LIN {X 0,Y 372.298,Z 1147.138,A -85,B 0,C 180,E1 19316.898,E2 19316.898} C_VEL
LIN {X 0,Y 364.057,Z 1169.224,A -85,B 0,C 180,E1 19324.16,E2 19324.16} C_VEL
LIN {X 0,Y 359.69,Z 1184.497,A -85,B 0,C 180,E1 19331.078,E2 19331.078} C_VEL
LIN {X 0,Y 357.708,Z 1194.571,A -85,B 0,C 180,E1 19337.805,E2 19337.805} C_VEL
LIN {X 0,Y 357.23,Z 1199.163,A -85,B 0,C 180,E1 19342.708,E2 19342.708} C_VEL
LIN {X 0,Y 357.403,Z 1201.877,A -85,B 0,C 180,E1 19349.999,E2 19349.999} C_VEL
LIN {X 0,Y 357.158,Z 1200.648,A -85,B 0,C 180,E1 19354.853,E2 19354.853} C_VEL
LIN {X 0,Y 357.531,Z 1196.078,A -85,B 0,C 180,E1 19360.963,E2 19360.963} C_VEL
LIN {X 0,Y 359.366,Z 1186.13,A -85,B 0,C 180,E1 19368.221,E2 19368.221} C_VEL
LIN {X 0,Y 364.091,Z 1170.43,A -85,B 0,C 180,E1 19375.834,E2 19375.834} C_VEL
LIN {X 0,Y 373.501,Z 1147.076,A -85,B 0,C 180,E1 19383.764,E2 19383.764} C_VEL
LIN {X 0,Y 386.478,Z 1119.54,A -85,B 0,C 180,E1 19390.645,E2 19390.645} C_VEL
LIN {X 0,Y 403.357,Z 1085.357,A -85,B 0,C 180,E1 19396.93,E2 19396.93} C_VEL
LIN {X 0,Y 421.007,Z 1048.766,A -85,B 0,C 180,E1 19401.873,E2 19401.873} C_VEL
LIN {X 0,Y 428.353,Z 1032.866,A -85,B 0,C 180,E1 19403.602,E2 19403.602} C_VEL
LIN {X 0,Y 431.334,Z 1020.773,A -85,B 0,C 180,E1 19405.233,E2 19405.233} C_VEL
LIN {X 0,Y 434.515,Z 1008.135,A -85,B 0,C 180,E1 19406.804,E2 19406.804} C_VEL
LIN {X 0,Y 450.973,Z 967.222,A -85,B 0,C 180,E1 19409.773,E2 19409.773} C_VEL
LIN {X 0,Y 465.114,Z 924.641,A -85,B 0,C 180,E1 19412.061,E2 19412.061} C_VEL
LIN {X 0,Y 459.039,Z 904.432,A -85,B 0,C 180,E1 19416.015,E2 19416.015} C_VEL
LIN {X 0,Y 451.558,Z 885.268,A -85,B 0,C 180,E1 19420.962,E2 19420.962} C_VEL
LIN {X 0,Y 444.782,Z 870.029,A -85,B 0,C 180,E1 19426.623,E2 19426.623} C_VEL
LIN {X 0,Y 441.283,Z 863.474,A -85,B 0,C 180,E1 19430.644,E2 19430.644} C_VEL
LIN {X 0,Y 439.558,Z 858.068,A -85,B 0,C 180,E1 19435.075,E2 19435.075} C_VEL
LIN {X 0,Y 439.377,Z 858.667,A -85,B 0,C 180,E1 19441.299,E2 19441.299} C_VEL
LIN {X 0,Y 441.594,Z 865.474,A -85,B 0,C 180,E1 19446.576,E2 19446.576} C_VEL
LIN {X 0,Y 445.757,Z 876.264,A -85,B 0,C 180,E1 19451.742,E2 19451.742} C_VEL
LIN {X 0,Y 451.62,Z 892.448,A -85,B 0,C 180,E1 19457.03,E2 19457.03} C_VEL
LIN {X 0,Y 457.495,Z 912.755,A -85,B 0,C 180,E1 19461.942,E2 19461.942} C_VEL
LIN {X 0,Y 459.188,Z 923.225,A -85,B 0,C 180,E1 19463.947,E2 19463.947} C_VEL
LIN {X 0,Y 443.527,Z 964.309,A -85,B 0,C 180,E1 19466.729,E2 19466.729} C_VEL
LIN {X 0,Y 425.31,Z 1003.875,A -85,B 0,C 180,E1 19470.42,E2 19470.42} C_VEL
LIN {X 0,Y 407.151,Z 1038.144,A -85,B 0,C 180,E1 19474.868,E2 19474.868} C_VEL
LIN {X 0,Y 390.184,Z 1067.744,A -85,B 0,C 180,E1 19480.105,E2 19480.105} C_VEL
LIN {X 0,Y 374.283,Z 1094.174,A -85,B 0,C 180,E1 19486.659,E2 19486.659} C_VEL
LIN {X 0,Y 362.655,Z 1114.122,A -85,B 0,C 180,E1 19493.626,E2 19493.626} C_VEL
LIN {X 0,Y 355.097,Z 1129.056,A -85,B 0,C 180,E1 19501.232,E2 19501.232} C_VEL
LIN {X 0,Y 351.155,Z 1138.273,A -85,B 0,C 180,E1 19508.598,E2 19508.598} C_VEL
LIN {X 0,Y 349.591,Z 1142.566,A -85,B 0,C 180,E1 19514.97,E2 19514.97} C_VEL
LIN {X 0,Y 349.351,Z 1143.375,A -85,B 0,C 180,E1 19522.545,E2 19522.545} C_VEL
LIN {X 0,Y 350.426,Z 1139.643,A -85,B 0,C 180,E1 19530.001,E2 19530.001} C_VEL
LIN {X 0,Y 352.724,Z 1131.212,A -85,B 0,C 180,E1 19537.386,E2 19537.386} C_VEL
LIN {X 0,Y 357.711,Z 1118.01,A -85,B 0,C 180,E1 19544.684,E2 19544.684} C_VEL
LIN {X 0,Y 366.523,Z 1099.034,A -85,B 0,C 180,E1 19551.782,E2 19551.782} C_VEL
LIN {X 0,Y 378.822,Z 1074.876,A -85,B 0,C 180,E1 19558.276,E2 19558.276} C_VEL
LIN {X 0,Y 394.375,Z 1044.03,A -85,B 0,C 180,E1 19564.249,E2 19564.249} C_VEL
LIN {X 0,Y 410.276,Z 1010.143,A -85,B 0,C 180,E1 19569.011,E2 19569.011} C_VEL
LIN {X 0,Y 425.898,Z 973.002,A -85,B 0,C 180,E1 19572.877,E2 19572.877} C_VEL
LIN {X 0,Y 441.528,Z 928.725,A -85,B 0,C 180,E1 19576.199,E2 19576.199} C_VEL
LIN {X 0,Y 445.75,Z 914.752,A -85,B 0,C 180,E1 19577.03,E2 19577.03} C_VEL
LIN {X 0,Y 437.347,Z 885.924,A -85,B 0,C 180,E1 19581.941,E2 19581.941} C_VEL
LIN {X 0,Y 428.04,Z 862.19,A -85,B 0,C 180,E1 19586.817,E2 19586.817} C_VEL
LIN {X 0,Y 417.98,Z 841.816,A -85,B 0,C 180,E1 19592.252,E2 19592.252} C_VEL
LIN {X 0,Y 410.472,Z 828.721,A -85,B 0,C 180,E1 19596.981,E2 19596.981} C_VEL
LIN {X 0,Y 406.667,Z 822.607,A -85,B 0,C 180,E1 19599.89,E2 19599.89} C_VEL
LIN {X 0,Y 403.865,Z 817.713,A -85,B 0,C 180,E1 19602.576,E2 19602.576} C_VEL
LIN {X 0,Y 400.692,Z 811.484,A -85,B 0,C 180,E1 19607.241,E2 19607.241} C_VEL
LIN {X 0,Y 399.55,Z 810.186,A -85,B 0,C 180,E1 19615.656,E2 19615.656} C_VEL
LIN {X 0,Y 402.264,Z 812.631,A -85,B 0,C 180,E1 19620.532,E2 19620.532} C_VEL
LIN {X 0,Y 406.945,Z 820.695,A -85,B 0,C 180,E1 19625.454,E2 19625.454} C_VEL
LIN {X 0,Y 414.067,Z 831.922,A -85,B 0,C 180,E1 19630.382,E2 19630.382} C_VEL
LIN {X 0,Y 424.174,Z 849.805,A -85,B 0,C 180,E1 19635.792,E2 19635.792} C_VEL
LIN {X 0,Y 435.914,Z 873.631,A -85,B 0,C 180,E1 19641.105,E2 19641.105} C_VEL
LIN {X 0,Y 447.798,Z 903.771,A -85,B 0,C 180,E1 19646.285,E2 19646.285} C_VEL
LIN {X 0,Y 453.221,Z 922.428,A -85,B 0,C 180,E1 19648.947,E2 19648.947} C_VEL
LIN {X 0,Y 439.542,Z 968.645,A -85,B 0,C 180,E1 19651.454,E2 19651.454} C_VEL
LIN {X 0,Y 424.425,Z 1010.952,A -85,B 0,C 180,E1 19654.623,E2 19654.623} C_VEL
LIN {X 0,Y 407,Z 1053.443,A -85,B 0,C 180,E1 19658.985,E2 19658.985} C_VEL
LIN {X 0,Y 391.108,Z 1089.121,A -85,B 0,C 180,E1 19663.978,E2 19663.978} C_VEL
LIN {X 0,Y 376.256,Z 1121.494,A -85,B 0,C 180,E1 19670.013,E2 19670.013} C_VEL
LIN {X 0,Y 364.257,Z 1148.631,A -85,B 0,C 180,E1 19676.893,E2 19676.893} C_VEL
LIN {X 0,Y 356.026,Z 1170.188,A -85,B 0,C 180,E1 19684.276,E2 19684.276} C_VEL
LIN {X 0,Y 351.536,Z 1185.408,A -85,B 0,C 180,E1 19691.659,E2 19691.659} C_VEL
LIN {X 0,Y 349.74,Z 1195.19,A -85,B 0,C 180,E1 19698.787,E2 19698.787} C_VEL
LIN {X 0,Y 349.272,Z 1199.924,A -85,B 0,C 180,E1 19705.035,E2 19705.035} C_VEL
LIN {X 0,Y 349.526,Z 1201.22,A -85,B 0,C 180,E1 19709.999,E2 19709.999} C_VEL
LIN {X 0,Y 349.229,Z 1199.679,A -85,B 0,C 180,E1 19715.66,E2 19715.66} C_VEL
LIN {X 0,Y 349.823,Z 1194.118,A -85,B 0,C 180,E1 19722.472,E2 19722.472} C_VEL
LIN {X 0,Y 352.296,Z 1183.154,A -85,B 0,C 180,E1 19730.068,E2 19730.068} C_VEL
LIN {X 0,Y 357.852,Z 1166.625,A -85,B 0,C 180,E1 19737.677,E2 19737.677} C_VEL
LIN {X 0,Y 368.006,Z 1143.362,A -85,B 0,C 180,E1 19745.45,E2 19745.45} C_VEL
LIN {X 0,Y 381.934,Z 1115.333,A -85,B 0,C 180,E1 19752.267,E2 19752.267} C_VEL
LIN {X 0,Y 399.336,Z 1081.94,A -85,B 0,C 180,E1 19758.284,E2 19758.284} C_VEL
LIN {X 0,Y 417.911,Z 1044.442,A -85,B 0,C 180,E1 19763.226,E2 19763.226} C_VEL
LIN {X 0,Y 434.515,Z 1008.135,A -85,B 0,C 180,E1 19766.804,E2 19766.804} C_VEL
LIN {X 0,Y 435.747,Z 999.983,A -85,B 0,C 180,E1 19767.933,E2 19767.933} C_VEL
LIN {X 0,Y 437.139,Z 991.635,A -85,B 0,C 180,E1 19769.014,E2 19769.014} C_VEL
LIN {X 0,Y 454.038,Z 947.387,A -85,B 0,C 180,E1 19771.825,E2 19771.825} C_VEL
LIN {X 0,Y 460.132,Z 928.064,A -85,B 0,C 180,E1 19772.848,E2 19772.848} C_VEL
LIN {X 0,Y 454.249,Z 907.989,A -85,B 0,C 180,E1 19776.996,E2 19776.996} C_VEL
LIN {X 0,Y 447.608,Z 890.491,A -85,B 0,C 180,E1 19781.808,E2 19781.808} C_VEL
LIN {X 0,Y 441.752,Z 876.873,A -85,B 0,C 180,E1 19787.158,E2 19787.158} C_VEL
LIN {X 0,Y 438.637,Z 870.605,A -85,B 0,C 180,E1 19791.212,E2 19791.212} C_VEL
LIN {X 0,Y 437.371,Z 865.682,A -85,B 0,C 180,E1 19795.05,E2 19795.05} C_VEL
LIN {X 0,Y 437.168,Z 865.729,A -85,B 0,C 180,E1 19800.872,E2 19800.872} C_VEL
LIN {X 0,Y 439.014,Z 873.18,A -85,B 0,C 180,E1 19806.615,E2 19806.615} C_VEL
LIN {X 0,Y 443.01,Z 884.158,A -85,B 0,C 180,E1 19811.816,E2 19811.816} C_VEL
LIN {X 0,Y 448.428,Z 900.54,A -85,B 0,C 180,E1 19817.155,E2 19817.155} C_VEL
LIN {X 0,Y 453.305,Z 919.811,A -85,B 0,C 180,E1 19821.836,E2 19821.836} C_VEL
LIN {X 0,Y 454.599,Z 925.88,A -85,B 0,C 180,E1 19823.12,E2 19823.12} C_VEL
LIN {X 0,Y 438.258,Z 967.608,A -85,B 0,C 180,E1 19826.048,E2 19826.048} C_VEL
LIN {X 0,Y 420.056,Z 1005.918,A -85,B 0,C 180,E1 19829.672,E2 19829.672} C_VEL
LIN {X 0,Y 400.332,Z 1041.744,A -85,B 0,C 180,E1 19834.425,E2 19834.425} C_VEL
LIN {X 0,Y 382.656,Z 1071.18,A -85,B 0,C 180,E1 19839.854,E2 19839.854} C_VEL
LIN {X 0,Y 366.795,Z 1096.673,A -85,B 0,C 180,E1 19846.409,E2 19846.409} C_VEL
LIN {X 0,Y 355.017,Z 1115.873,A -85,B 0,C 180,E1 19853.424,E2 19853.424} C_VEL
LIN {X 0,Y 347.124,Z 1130.81,A -85,B 0,C 180,E1 19861.39,E2 19861.39} C_VEL
LIN {X 0,Y 343.082,Z 1139.88,A -85,B 0,C 180,E1 19869.369,E2 19869.369} C_VEL
LIN {X 0,Y 341.489,Z 1144.054,A -85,B 0,C 180,E1 19877.218,E2 19877.218} C_VEL
LIN {X 0,Y 341.718,Z 1143.309,A -85,B 0,C 180,E1 19884.927,E2 19884.927} C_VEL
LIN {X 0,Y 342.88,Z 1139.282,A -85,B 0,C 180,E1 19891.264,E2 19891.264} C_VEL
LIN {X 0,Y 345.586,Z 1130.291,A -85,B 0,C 180,E1 19898.805,E2 19898.805} C_VEL
LIN {X 0,Y 351.36,Z 1116.165,A -85,B 0,C 180,E1 19906.235,E2 19906.235} C_VEL
LIN {X 0,Y 361.614,Z 1095.823,A -85,B 0,C 180,E1 19913.62,E2 19913.62} C_VEL
LIN {X 0,Y 376.074,Z 1068.411,A -85,B 0,C 180,E1 19920.552,E2 19920.552} C_VEL
LIN {X 0,Y 391.531,Z 1038.192,A -85,B 0,C 180,E1 19926.058,E2 19926.058} C_VEL
LIN {X 0,Y 408.575,Z 1002.491,A -85,B 0,C 180,E1 19930.799,E2 19930.799} C_VEL
LIN {X 0,Y 425.037,Z 962.822,A -85,B 0,C 180,E1 19934.608,E2 19934.608} C_VEL
LIN {X 0,Y 438.935,Z 922.777,A -85,B 0,C 180,E1 19937.426,E2 19937.426} C_VEL
LIN {X 0,Y 439.949,Z 917.005,A -85,B 0,C 180,E1 19937.907,E2 19937.907} C_VEL
LIN {X 0,Y 432.477,Z 890.045,A -85,B 0,C 180,E1 19942.663,E2 19942.663} C_VEL
LIN {X 0,Y 423.57,Z 866.773,A -85,B 0,C 180,E1 19947.639,E2 19947.639} C_VEL
LIN {X 0,Y 414.395,Z 847.583,A -85,B 0,C 180,E1 19952.992,E2 19952.992} C_VEL
LIN {X 0,Y 407.812,Z 835.438,A -85,B 0,C 180,E1 19957.505,E2 19957.505} C_VEL
LIN {X 0,Y 402.53,Z 825.678,A -85,B 0,C 180,E1 19962.396,E2 19962.396} C_VEL
LIN {X 0,Y 399.093,Z 819.165,A -85,B 0,C 180,E1 19967.418,E2 19967.418} C_VEL
LIN {X 0,Y 398.181,Z 817.941,A -85,B 0,C 180,E1 19975.641,E2 19975.641} C_VEL
LIN {X 0,Y 400.691,Z 820.234,A -85,B 0,C 180,E1 19980.332,E2 19980.332} C_VEL
LIN {X 0,Y 405.241,Z 828.467,A -85,B 0,C 180,E1 19985.343,E2 19985.343} C_VEL
LIN {X 0,Y 411.935,Z 839.468,A -85,B 0,C 180,E1 19990.163,E2 19990.163} C_VEL
LIN {X 0,Y 421.528,Z 857.101,A -85,B 0,C 180,E1 19995.546,E2 19995.546} C_VEL
LIN {X 0,Y 432.262,Z 880.049,A -85,B 0,C 180,E1 20000.724,E2 20000.724} C_VEL
LIN {X 0,Y 442.967,Z 908.697,A -85,B 0,C 180,E1 20005.777,E2 20005.777} C_VEL
LIN {X 0,Y 447.647,Z 925.803,A -85,B 0,C 180,E1 20008.28,E2 20008.28} C_VEL
LIN {X 0,Y 434.055,Z 970.322,A -85,B 0,C 180,E1 20010.742,E2 20010.742} C_VEL
LIN {X 0,Y 418.224,Z 1012.969,A -85,B 0,C 180,E1 20013.996,E2 20013.996} C_VEL
LIN {X 0,Y 400.743,Z 1054.371,A -85,B 0,C 180,E1 20018.319,E2 20018.319} C_VEL
LIN {X 0,Y 383.631,Z 1091.344,A -85,B 0,C 180,E1 20023.632,E2 20023.632} C_VEL
LIN {X 0,Y 368.518,Z 1123.103,A -85,B 0,C 180,E1 20029.77,E2 20029.77} C_VEL
LIN {X 0,Y 355.85,Z 1150.918,A -85,B 0,C 180,E1 20037.127,E2 20037.127} C_VEL
LIN {X 0,Y 347.601,Z 1171.912,A -85,B 0,C 180,E1 20044.813,E2 20044.813} C_VEL
LIN {X 0,Y 343.236,Z 1187.034,A -85,B 0,C 180,E1 20052.711,E2 20052.711} C_VEL
LIN {X 0,Y 341.724,Z 1195.789,A -85,B 0,C 180,E1 20059.81,E2 20059.81} C_VEL
LIN {X 0,Y 341.456,Z 1200.202,A -85,B 0,C 180,E1 20067.462,E2 20067.462} C_VEL
LIN {X 0,Y 341.586,Z 1200.233,A -85,B 0,C 180,E1 20072.534,E2 20072.534} C_VEL
LIN {X 0,Y 341.687,Z 1196.101,A -85,B 0,C 180,E1 20080.188,E2 20080.188} C_VEL
LIN {X 0,Y 343.45,Z 1186.747,A -85,B 0,C 180,E1 20087.937,E2 20087.937} C_VEL
LIN {X 0,Y 348.573,Z 1170.894,A -85,B 0,C 180,E1 20096.29,E2 20096.29} C_VEL
LIN {X 0,Y 358.125,Z 1149.375,A -85,B 0,C 180,E1 20104.223,E2 20104.223} C_VEL
LIN {X 0,Y 372.851,Z 1120.635,A -85,B 0,C 180,E1 20111.882,E2 20111.882} C_VEL
LIN {X 0,Y 390.029,Z 1088.483,A -85,B 0,C 180,E1 20118.07,E2 20118.07} C_VEL
LIN {X 0,Y 409.11,Z 1052.094,A -85,B 0,C 180,E1 20123.231,E2 20123.231} C_VEL
LIN {X 0,Y 429.335,Z 1009.589,A -85,B 0,C 180,E1 20127.571,E2 20127.571} C_VEL
LIN {X 0,Y 437.139,Z 991.635,A -85,B 0,C 180,E1 20129.014,E2 20129.014} C_VEL
LIN {X 0,Y 440.785,Z 978.212,A -85,B 0,C 180,E1 20130.407,E2 20130.407} C_VEL
LIN {X 0,Y 444.102,Z 964.397,A -85,B 0,C 180,E1 20131.741,E2 20131.741} C_VEL
LIN {X 0,Y 455.353,Z 932.19,A -85,B 0,C 180,E1 20133.536,E2 20133.536} C_VEL
LIN {X 0,Y 449.837,Z 912.417,A -85,B 0,C 180,E1 20137.8,E2 20137.8} C_VEL
LIN {X 0,Y 443.79,Z 895.75,A -85,B 0,C 180,E1 20142.62,E2 20142.62} C_VEL
LIN {X 0,Y 438.305,Z 882.887,A -85,B 0,C 180,E1 20148.067,E2 20148.067} C_VEL
LIN {X 0,Y 436.988,Z 879.284,A -85,B 0,C 180,E1 20150.049,E2 20150.049} C_VEL
LIN {X 0,Y 434.727,Z 873.097,A -85,B 0,C 180,E1 20156.019,E2 20156.019} C_VEL
LIN {X 0,Y 434.664,Z 873.589,A -85,B 0,C 180,E1 20161.002,E2 20161.002} C_VEL
LIN {X 0,Y 436.602,Z 881.447,A -85,B 0,C 180,E1 20166.964,E2 20166.964} C_VEL
LIN {X 0,Y 440.476,Z 893.236,A -85,B 0,C 180,E1 20172.387,E2 20172.387} C_VEL
LIN {X 0,Y 445.54,Z 910.373,A -85,B 0,C 180,E1 20177.779,E2 20177.779} C_VEL
LIN {X 0,Y 449.726,Z 929.919,A -85,B 0,C 180,E1 20182.394,E2 20182.394} C_VEL
LIN {X 0,Y 432.01,Z 973.227,A -85,B 0,C 180,E1 20185.539,E2 20185.539} C_VEL
LIN {X 0,Y 413.804,Z 1009.781,A -85,B 0,C 180,E1 20189.127,E2 20189.127} C_VEL
LIN {X 0,Y 393.687,Z 1045.079,A -85,B 0,C 180,E1 20193.925,E2 20193.925} C_VEL
LIN {X 0,Y 374.913,Z 1074.943,A -85,B 0,C 180,E1 20199.665,E2 20199.665} C_VEL
LIN {X 0,Y 359.807,Z 1098.302,A -85,B 0,C 180,E1 20205.893,E2 20205.893} C_VEL
LIN {X 0,Y 346.94,Z 1118.402,A -85,B 0,C 180,E1 20213.565,E2 20213.565} C_VEL
LIN {X 0,Y 339.767,Z 1131.284,A -85,B 0,C 180,E1 20220.712,E2 20220.712} C_VEL
LIN {X 0,Y 335.363,Z 1140.424,A -85,B 0,C 180,E1 20228.872,E2 20228.872} C_VEL
LIN {X 0,Y 333.656,Z 1144.679,A -85,B 0,C 180,E1 20236.913,E2 20236.913} C_VEL
LIN {X 0,Y 333.835,Z 1143.99,A -85,B 0,C 180,E1 20244.871,E2 20244.871} C_VEL
LIN {X 0,Y 335.028,Z 1140.06,A -85,B 0,C 180,E1 20251.294,E2 20251.294} C_VEL
LIN {X 0,Y 337.826,Z 1131.151,A -85,B 0,C 180,E1 20259.008,E2 20259.008} C_VEL
LIN {X 0,Y 343.861,Z 1117.149,A -85,B 0,C 180,E1 20266.599,E2 20266.599} C_VEL
LIN {X 0,Y 354.073,Z 1097.564,A -85,B 0,C 180,E1 20273.92,E2 20273.92} C_VEL
LIN {X 0,Y 367.729,Z 1072.531,A -85,B 0,C 180,E1 20280.532,E2 20280.532} C_VEL
LIN {X 0,Y 383.67,Z 1042.925,A -85,B 0,C 180,E1 20286.215,E2 20286.215} C_VEL
LIN {X 0,Y 401.682,Z 1006.468,A -85,B 0,C 180,E1 20291.243,E2 20291.243} C_VEL
LIN {X 0,Y 417.381,Z 970.33,A -85,B 0,C 180,E1 20294.875,E2 20294.875} C_VEL
LIN {X 0,Y 433.244,Z 927.056,A -85,B 0,C 180,E1 20298.059,E2 20298.059} C_VEL
LIN {X 0,Y 434.663,Z 921.259,A -85,B 0,C 180,E1 20298.476,E2 20298.476} C_VEL
LIN {X 0,Y 427.695,Z 894.542,A -85,B 0,C 180,E1 20303.349,E2 20303.349} C_VEL
LIN {X 0,Y 419.208,Z 871.284,A -85,B 0,C 180,E1 20308.48,E2 20308.48} C_VEL
LIN {X 0,Y 409.774,Z 850.757,A -85,B 0,C 180,E1 20314.535,E2 20314.535} C_VEL
LIN {X 0,Y 403.123,Z 838.446,A -85,B 0,C 180,E1 20319.806,E2 20319.806} C_VEL
LIN {X 0,Y 399.952,Z 832.552,A -85,B 0,C 180,E1 20323.261,E2 20323.261} C_VEL
LIN {X 0,Y 397.62,Z 826.94,A -85,B 0,C 180,E1 20327.371,E2 20327.371} C_VEL
LIN {X 0,Y 396.681,Z 825.691,A -85,B 0,C 180,E1 20335.624,E2 20335.624} C_VEL
LIN {X 0,Y 399.061,Z 828.056,A -85,B 0,C 180,E1 20340.208,E2 20340.208} C_VEL
LIN {X 0,Y 403.293,Z 835.821,A -85,B 0,C 180,E1 20345.032,E2 20345.032} C_VEL
LIN {X 0,Y 409.418,Z 846.53,A -85,B 0,C 180,E1 20349.823,E2 20349.823} C_VEL
LIN {X 0,Y 418.491,Z 864.046,A -85,B 0,C 180,E1 20355.238,E2 20355.238} C_VEL
LIN {X 0,Y 428.465,Z 886.467,A -85,B 0,C 180,E1 20360.376,E2 20360.376} C_VEL
LIN {X 0,Y 438.653,Z 915.128,A -85,B 0,C 180,E1 20365.501,E2 20365.501} C_VEL
LIN {X 0,Y 442.302,Z 928.026,A -85,B 0,C 180,E1 20367.514,E2 20367.514} C_VEL
LIN {X 0,Y 428.363,Z 972.775,A -85,B 0,C 180,E1 20370.058,E2 20370.058} C_VEL
LIN {X 0,Y 411.337,Z 1016.852,A -85,B 0,C 180,E1 20373.528,E2 20373.528} C_VEL
LIN {X 0,Y 393.953,Z 1056.364,A -85,B 0,C 180,E1 20377.775,E2 20377.775} C_VEL
LIN {X 0,Y 376.276,Z 1093.339,A -85,B 0,C 180,E1 20383.232,E2 20383.232} C_VEL
LIN {X 0,Y 361.11,Z 1124.016,A -85,B 0,C 180,E1 20389.366,E2 20389.366} C_VEL
LIN {X 0,Y 348.271,Z 1151.29,A -85,B 0,C 180,E1 20396.783,E2 20396.783} C_VEL
LIN {X 0,Y 340.042,Z 1171.302,A -85,B 0,C 180,E1 20404.322,E2 20404.322} C_VEL
LIN {X 0,Y 335.469,Z 1186.262,A -85,B 0,C 180,E1 20412.297,E2 20412.297} C_VEL
LIN {X 0,Y 333.852,Z 1195.074,A -85,B 0,C 180,E1 20419.568,E2 20419.568} C_VEL
LIN {X 0,Y 333.57,Z 1199.545,A -85,B 0,C 180,E1 20427.402,E2 20427.402} C_VEL
LIN {X 0,Y 333.694,Z 1199.587,A -85,B 0,C 180,E1 20432.594,E2 20432.594} C_VEL
LIN {X 0,Y 333.803,Z 1195.472,A -85,B 0,C 180,E1 20440.431,E2 20440.431} C_VEL
LIN {X 0,Y 335.706,Z 1186.151,A -85,B 0,C 180,E1 20448.365,E2 20448.365} C_VEL
LIN {X 0,Y 340.633,Z 1171.567,A -85,B 0,C 180,E1 20456.334,E2 20456.334} C_VEL
LIN {X 0,Y 349.937,Z 1151.511,A -85,B 0,C 180,E1 20464.15,E2 20464.15} C_VEL
LIN {X 0,Y 364.606,Z 1123.772,A -85,B 0,C 180,E1 20471.894,E2 20471.894} C_VEL
LIN {X 0,Y 382.005,Z 1092.753,A -85,B 0,C 180,E1 20478.209,E2 20478.209} C_VEL
LIN {X 0,Y 402.627,Z 1054.801,A -85,B 0,C 180,E1 20483.795,E2 20483.795} C_VEL
LIN {X 0,Y 422.262,Z 1015.331,A -85,B 0,C 180,E1 20487.97,E2 20487.97} C_VEL
LIN {X 0,Y 440.817,Z 972.947,A -85,B 0,C 180,E1 20491.21,E2 20491.21} C_VEL
LIN {X 0,Y 444.102,Z 964.397,A -85,B 0,C 180,E1 20491.741,E2 20491.741} C_VEL
LIN {X 0,Y 448.813,Z 949.442,A -85,B 0,C 180,E1 20492.813,E2 20492.813} C_VEL
LIN {X 0,Y 450.391,Z 936.31,A -85,B 0,C 180,E1 20494.285,E2 20494.285} C_VEL
LIN {X 0,Y 445.385,Z 916.928,A -85,B 0,C 180,E1 20498.614,E2 20498.614} C_VEL
LIN {X 0,Y 439.799,Z 900.879,A -85,B 0,C 180,E1 20503.487,E2 20503.487} C_VEL
LIN {X 0,Y 435.77,Z 890.558,A -85,B 0,C 180,E1 20507.996,E2 20507.996} C_VEL
LIN {X 0,Y 433.138,Z 884.863,A -85,B 0,C 180,E1 20511.983,E2 20511.983} C_VEL
LIN {X 0,Y 432.186,Z 880.636,A -85,B 0,C 180,E1 20515.996,E2 20515.996} C_VEL
LIN {X 0,Y 432.089,Z 881.213,A -85,B 0,C 180,E1 20521.008,E2 20521.008} C_VEL
LIN {X 0,Y 433.788,Z 889.019,A -85,B 0,C 180,E1 20527.009,E2 20527.009} C_VEL
LIN {X 0,Y 437.424,Z 901.023,A -85,B 0,C 180,E1 20532.475,E2 20532.475} C_VEL
LIN {X 0,Y 441.708,Z 917.444,A -85,B 0,C 180,E1 20537.656,E2 20537.656} C_VEL
LIN {X 0,Y 444.85,Z 934.711,A -85,B 0,C 180,E1 20541.817,E2 20541.817} C_VEL
LIN {X 0,Y 426.821,Z 976.648,A -85,B 0,C 180,E1 20544.839,E2 20544.839} C_VEL
LIN {X 0,Y 407.57,Z 1013.666,A -85,B 0,C 180,E1 20548.568,E2 20548.568} C_VEL
LIN {X 0,Y 387.932,Z 1046.943,A -85,B 0,C 180,E1 20553.185,E2 20553.185} C_VEL
LIN {X 0,Y 368.056,Z 1077.361,A -85,B 0,C 180,E1 20559.16,E2 20559.16} C_VEL
LIN {X 0,Y 352.488,Z 1100.34,A -85,B 0,C 180,E1 20565.517,E2 20565.517} C_VEL
LIN {X 0,Y 339.415,Z 1119.989,A -85,B 0,C 180,E1 20573.276,E2 20573.276} C_VEL
LIN {X 0,Y 331.338,Z 1133.583,A -85,B 0,C 180,E1 20581.39,E2 20581.39} C_VEL
LIN {X 0,Y 327.695,Z 1140.968,A -85,B 0,C 180,E1 20588.353,E2 20588.353} C_VEL
LIN {X 0,Y 325.795,Z 1145.367,A -85,B 0,C 180,E1 20596.955,E2 20596.955} C_VEL
LIN {X 0,Y 325.92,Z 1144.724,A -85,B 0,C 180,E1 20604.681,E2 20604.681} C_VEL
LIN {X 0,Y 327.188,Z 1140.837,A -85,B 0,C 180,E1 20611.325,E2 20611.325} C_VEL
LIN {X 0,Y 330.096,Z 1132.003,A -85,B 0,C 180,E1 20619.221,E2 20619.221} C_VEL
LIN {X 0,Y 336.348,Z 1118.138,A -85,B 0,C 180,E1 20626.981,E2 20626.981} C_VEL
LIN {X 0,Y 346.944,Z 1098.638,A -85,B 0,C 180,E1 20634.444,E2 20634.444} C_VEL
LIN {X 0,Y 361.125,Z 1073.642,A -85,B 0,C 180,E1 20641.188,E2 20641.188} C_VEL
LIN {X 0,Y 377.447,Z 1044.355,A -85,B 0,C 180,E1 20646.909,E2 20646.909} C_VEL
LIN {X 0,Y 395.856,Z 1008.158,A -85,B 0,C 180,E1 20651.97,E2 20651.97} C_VEL
LIN {X 0,Y 412.103,Z 971.95,A -85,B 0,C 180,E1 20655.655,E2 20655.655} C_VEL
LIN {X 0,Y 428.557,Z 928.256,A -85,B 0,C 180,E1 20658.884,E2 20658.884} C_VEL
LIN {X 0,Y 429.331,Z 925.06,A -85,B 0,C 180,E1 20659.134,E2 20659.134} C_VEL
LIN {X 0,Y 423.055,Z 899.725,A -85,B 0,C 180,E1 20663.88,E2 20663.88} C_VEL
LIN {X 0,Y 415.512,Z 877.431,A -85,B 0,C 180,E1 20668.946,E2 20668.946} C_VEL
LIN {X 0,Y 406.688,Z 857.32,A -85,B 0,C 180,E1 20675.037,E2 20675.037} C_VEL
LIN {X 0,Y 400.812,Z 845.659,A -85,B 0,C 180,E1 20680.158,E2 20680.158} C_VEL
LIN {X 0,Y 397.955,Z 840.105,A -85,B 0,C 180,E1 20683.411,E2 20683.411} C_VEL
LIN {X 0,Y 395.639,Z 834.469,A -85,B 0,C 180,E1 20687.867,E2 20687.867} C_VEL
LIN {X 0,Y 395.316,Z 833.614,A -85,B 0,C 180,E1 20696.207,E2 20696.207} C_VEL
LIN {X 0,Y 397.334,Z 835.775,A -85,B 0,C 180,E1 20700.066,E2 20700.066} C_VEL
LIN {X 0,Y 401.176,Z 843.382,A -85,B 0,C 180,E1 20704.856,E2 20704.856} C_VEL
LIN {X 0,Y 407.172,Z 854.232,A -85,B 0,C 180,E1 20709.676,E2 20709.676} C_VEL
LIN {X 0,Y 415.57,Z 871.287,A -85,B 0,C 180,E1 20715.01,E2 20715.01} C_VEL
LIN {X 0,Y 425.149,Z 894.141,A -85,B 0,C 180,E1 20720.271,E2 20720.271} C_VEL
LIN {X 0,Y 434.473,Z 922.544,A -85,B 0,C 180,E1 20725.398,E2 20725.398} C_VEL
LIN {X 0,Y 436.687,Z 932.573,A -85,B 0,C 180,E1 20726.903,E2 20726.903} C_VEL
LIN {X 0,Y 422.714,Z 975.019,A -85,B 0,C 180,E1 20729.359,E2 20729.359} C_VEL
LIN {X 0,Y 405.188,Z 1018.977,A -85,B 0,C 180,E1 20732.878,E2 20732.878} C_VEL
LIN {X 0,Y 387.772,Z 1057.184,A -85,B 0,C 180,E1 20737.069,E2 20737.069} C_VEL
LIN {X 0,Y 369.562,Z 1094.076,A -85,B 0,C 180,E1 20742.605,E2 20742.605} C_VEL
LIN {X 0,Y 353.972,Z 1124.429,A -85,B 0,C 180,E1 20748.827,E2 20748.827} C_VEL
LIN {X 0,Y 340.81,Z 1151.385,A -85,B 0,C 180,E1 20756.34,E2 20756.34} C_VEL
LIN {X 0,Y 332.033,Z 1171.915,A -85,B 0,C 180,E1 20764.381,E2 20764.381} C_VEL
LIN {X 0,Y 327.492,Z 1186.538,A -85,B 0,C 180,E1 20772.545,E2 20772.545} C_VEL
LIN {X 0,Y 325.982,Z 1194.353,A -85,B 0,C 180,E1 20779.313,E2 20779.313} C_VEL
LIN {X 0,Y 325.707,Z 1198.888,A -85,B 0,C 180,E1 20787.339,E2 20787.339} C_VEL
LIN {X 0,Y 325.822,Z 1198.943,A -85,B 0,C 180,E1 20792.657,E2 20792.657} C_VEL
LIN {X 0,Y 325.924,Z 1194.845,A -85,B 0,C 180,E1 20800.686,E2 20800.686} C_VEL
LIN {X 0,Y 327.455,Z 1187.456,A -85,B 0,C 180,E1 20807.454,E2 20807.454} C_VEL
LIN {X 0,Y 332.047,Z 1173.866,A -85,B 0,C 180,E1 20815.615,E2 20815.615} C_VEL
LIN {X 0,Y 342.046,Z 1152.823,A -85,B 0,C 180,E1 20824.282,E2 20824.282} C_VEL
LIN {X 0,Y 356.258,Z 1127.047,A -85,B 0,C 180,E1 20831.881,E2 20831.881} C_VEL
LIN {X 0,Y 374.695,Z 1095.485,A -85,B 0,C 180,E1 20838.607,E2 20838.607} C_VEL
LIN {X 0,Y 394.502,Z 1060.417,A -85,B 0,C 180,E1 20844.001,E2 20844.001} C_VEL
LIN {X 0,Y 414.889,Z 1021.729,A -85,B 0,C 180,E1 20848.315,E2 20848.315} C_VEL
LIN {X 0,Y 433.305,Z 981.581,A -85,B 0,C 180,E1 20851.551,E2 20851.551} C_VEL
LIN {X 0,Y 449.972,Z 938.36,A -85,B 0,C 180,E1 20854.097,E2 20854.097} C_VEL
LIN {X 0,Y 450.391,Z 936.31,A -85,B 0,C 180,E1 20854.285,E2 20854.285} C_VEL
LIN {X 0,Y 448.638,Z 931.405,A -85,B 0,C 180,E1 20855.491,E2 20855.491} C_VEL
LIN {X 0,Y 441.977,Z 925.186,A -85,B 0,C 180,E1 20858.445,E2 20858.445} C_VEL
LIN {X 0,Y 436.794,Z 908.664,A -85,B 0,C 180,E1 20863.422,E2 20863.422} C_VEL
LIN {X 0,Y 432.235,Z 896.445,A -85,B 0,C 180,E1 20868.919,E2 20868.919} C_VEL
LIN {X 0,Y 429.643,Z 888.175,A -85,B 0,C 180,E1 20875.972,E2 20875.972} C_VEL
LIN {X 0,Y 429.408,Z 888.77,A -85,B 0,C 180,E1 20881.014,E2 20881.014} C_VEL
LIN {X 0,Y 430.875,Z 896.571,A -85,B 0,C 180,E1 20887.057,E2 20887.057} C_VEL
LIN {X 0,Y 434.138,Z 908.886,A -85,B 0,C 180,E1 20892.627,E2 20892.627} C_VEL
LIN {X 0,Y 437.757,Z 924.609,A -85,B 0,C 180,E1 20897.587,E2 20897.587} C_VEL
LIN {X 0,Y 440.015,Z 938.734,A -85,B 0,C 180,E1 20901.08,E2 20901.08} C_VEL
LIN {X 0,Y 421.578,Z 980.141,A -85,B 0,C 180,E1 20904.145,E2 20904.145} C_VEL
LIN {X 0,Y 401.599,Z 1017.16,A -85,B 0,C 180,E1 20907.943,E2 20907.943} C_VEL
LIN {X 0,Y 381.264,Z 1050.141,A -85,B 0,C 180,E1 20912.656,E2 20912.656} C_VEL
LIN {X 0,Y 361.579,Z 1079.284,A -85,B 0,C 180,E1 20918.524,E2 20918.524} C_VEL
LIN {X 0,Y 344.524,Z 1103.272,A -85,B 0,C 180,E1 20925.432,E2 20925.432} C_VEL
LIN {X 0,Y 331.836,Z 1121.638,A -85,B 0,C 180,E1 20933.001,E2 20933.001} C_VEL
LIN {X 0,Y 324.014,Z 1134.065,A -85,B 0,C 180,E1 20940.681,E2 20940.681} C_VEL
LIN {X 0,Y 319.483,Z 1142.627,A -85,B 0,C 180,E1 20949.224,E2 20949.224} C_VEL
LIN {X 0,Y 317.96,Z 1145.891,A -85,B 0,C 180,E1 20956.255,E2 20956.255} C_VEL
LIN {X 0,Y 318.035,Z 1145.429,A -85,B 0,C 180,E1 20964.548,E2 20964.548} C_VEL
LIN {X 0,Y 319.32,Z 1141.613,A -85,B 0,C 180,E1 20971.357,E2 20971.357} C_VEL
LIN {X 0,Y 322.341,Z 1132.858,A -85,B 0,C 180,E1 20979.445,E2 20979.445} C_VEL
LIN {X 0,Y 328.857,Z 1119.12,A -85,B 0,C 180,E1 20987.38,E2 20987.38} C_VEL
LIN {X 0,Y 340.963,Z 1097.89,A -85,B 0,C 180,E1 20995.603,E2 20995.603} C_VEL
LIN {X 0,Y 356.757,Z 1071.124,A -85,B 0,C 180,E1 21002.689,E2 21002.689} C_VEL
LIN {X 0,Y 373.884,Z 1040.845,A -85,B 0,C 180,E1 21008.421,E2 21008.421} C_VEL
LIN {X 0,Y 392.323,Z 1005.472,A -85,B 0,C 180,E1 21013.244,E2 21013.244} C_VEL
LIN {X 0,Y 410.003,Z 966.171,A -85,B 0,C 180,E1 21017.074,E2 21017.074} C_VEL
LIN {X 0,Y 423.938,Z 928.29,A -85,B 0,C 180,E1 21019.899,E2 21019.899} C_VEL
LIN {X 0,Y 418.142,Z 903.724,A -85,B 0,C 180,E1 21024.666,E2 21024.666} C_VEL
LIN {X 0,Y 410.946,Z 881.634,A -85,B 0,C 180,E1 21029.925,E2 21029.925} C_VEL
LIN {X 0,Y 403.447,Z 863.601,A -85,B 0,C 180,E1 21035.662,E2 21035.662} C_VEL
LIN {X 0,Y 398.189,Z 852.673,A -85,B 0,C 180,E1 21040.553,E2 21040.553} C_VEL
LIN {X 0,Y 395.726,Z 847.414,A -85,B 0,C 180,E1 21043.831,E2 21043.831} C_VEL
LIN {X 0,Y 393.818,Z 842.171,A -85,B 0,C 180,E1 21047.81,E2 21047.81} C_VEL
LIN {X 0,Y 393.435,Z 841.23,A -85,B 0,C 180,E1 21056.085,E2 21056.085} C_VEL
LIN {X 0,Y 395.366,Z 843.423,A -85,B 0,C 180,E1 21059.929,E2 21059.929} C_VEL
LIN {X 0,Y 399.061,Z 850.935,A -85,B 0,C 180,E1 21064.678,E2 21064.678} C_VEL
LIN {X 0,Y 404.676,Z 861.804,A -85,B 0,C 180,E1 21069.532,E2 21069.532} C_VEL
LIN {X 0,Y 411.87,Z 876.895,A -85,B 0,C 180,E1 21074.333,E2 21074.333} C_VEL
LIN {X 0,Y 420.818,Z 899.286,A -85,B 0,C 180,E1 21079.667,E2 21079.667} C_VEL
LIN {X 0,Y 429.634,Z 927.812,A -85,B 0,C 180,E1 21084.96,E2 21084.96} C_VEL
LIN {X 0,Y 431.491,Z 935.116,A -85,B 0,C 180,E1 21086.137,E2 21086.137} C_VEL
LIN {X 0,Y 416.218,Z 979.586,A -85,B 0,C 180,E1 21088.808,E2 21088.808} C_VEL
LIN {X 0,Y 399.098,Z 1021.106,A -85,B 0,C 180,E1 21092.21,E2 21092.21} C_VEL
LIN {X 0,Y 380.458,Z 1060.306,A -85,B 0,C 180,E1 21096.641,E2 21096.641} C_VEL
LIN {X 0,Y 362.123,Z 1096.189,A -85,B 0,C 180,E1 21102.207,E2 21102.207} C_VEL
LIN {X 0,Y 345.348,Z 1127.729,A -85,B 0,C 180,E1 21108.976,E2 21108.976} C_VEL
LIN {X 0,Y 332.887,Z 1152.371,A -85,B 0,C 180,E1 21116.213,E2 21116.213} C_VEL
LIN {X 0,Y 324.029,Z 1172.526,A -85,B 0,C 180,E1 21124.443,E2 21124.443} C_VEL
LIN {X 0,Y 319.736,Z 1185.759,A -85,B 0,C 180,E1 21132.108,E2 21132.108} C_VEL
LIN {X 0,Y 318.141,Z 1193.635,A -85,B 0,C 180,E1 21139.046,E2 21139.046} C_VEL
LIN {X 0,Y 317.837,Z 1198.231,A -85,B 0,C 180,E1 21147.274,E2 21147.274} C_VEL
LIN {X 0,Y 317.842,Z 1198.191,A -85,B 0,C 180,E1 21153.337,E2 21153.337} C_VEL
LIN {X 0,Y 318.051,Z 1194.22,A -85,B 0,C 180,E1 21160.954,E2 21160.954} C_VEL
LIN {X 0,Y 319.705,Z 1186.854,A -85,B 0,C 180,E1 21167.891,E2 21167.891} C_VEL
LIN {X 0,Y 324.618,Z 1173.31,A -85,B 0,C 180,E1 21176.245,E2 21176.245} C_VEL
LIN {X 0,Y 335.174,Z 1152.305,A -85,B 0,C 180,E1 21185.086,E2 21185.086} C_VEL
LIN {X 0,Y 349.015,Z 1128.423,A -85,B 0,C 180,E1 21192.34,E2 21192.34} C_VEL
LIN {X 0,Y 368.19,Z 1096.77,A -85,B 0,C 180,E1 21199.264,E2 21199.264} C_VEL
LIN {X 0,Y 387.694,Z 1063.759,A -85,B 0,C 180,E1 21204.506,E2 21204.506} C_VEL
LIN {X 0,Y 410.265,Z 1022.224,A -85,B 0,C 180,E1 21209.222,E2 21209.222} C_VEL
LIN {X 0,Y 428.649,Z 983.549,A -85,B 0,C 180,E1 21212.361,E2 21212.361} C_VEL
LIN {X 0,Y 445.695,Z 940.338,A -85,B 0,C 180,E1 21214.961,E2 21214.961} C_VEL
LIN {X 0,Y 441.977,Z 925.186,A -85,B 0,C 180,E1 21218.445,E2 21218.445} C_VEL
LIN {X 0,Y 439.143,Z 921.621,A -85,B 0,C 180,E1 21220.047,E2 21220.047} C_VEL
LIN {X 0,Y 434.052,Z 917.857,A -85,B 0,C 180,E1 21222.835,E2 21222.835} C_VEL
LIN {X 0,Y 430.077,Z 905.711,A -85,B 0,C 180,E1 21227.835,E2 21227.835} C_VEL
LIN {X 0,Y 427.009,Z 897.488,A -85,B 0,C 180,E1 21233.911,E2 21233.911} C_VEL
LIN {X 0,Y 426.782,Z 895.594,A -85,B 0,C 180,E1 21235.945,E2 21235.945} C_VEL
LIN {X 0,Y 426.57,Z 895.355,A -85,B 0,C 180,E1 21240.006,E2 21240.006} C_VEL
LIN {X 0,Y 427.538,Z 902.335,A -85,B 0,C 180,E1 21246.093,E2 21246.093} C_VEL
LIN {X 0,Y 430.112,Z 913.842,A -85,B 0,C 180,E1 21251.677,E2 21251.677} C_VEL
LIN {X 0,Y 433.256,Z 928.957,A -85,B 0,C 180,E1 21256.729,E2 21256.729} C_VEL
LIN {X 0,Y 435.221,Z 943.05,A -85,B 0,C 180,E1 21260.373,E2 21260.373} C_VEL
LIN {X 0,Y 416.407,Z 983.485,A -85,B 0,C 180,E1 21263.422,E2 21263.422} C_VEL
LIN {X 0,Y 395.699,Z 1020.575,A -85,B 0,C 180,E1 21267.283,E2 21267.283} C_VEL
LIN {X 0,Y 374.644,Z 1053.338,A -85,B 0,C 180,E1 21272.111,E2 21272.111} C_VEL
LIN {X 0,Y 354.92,Z 1081.503,A -85,B 0,C 180,E1 21277.936,E2 21277.936} C_VEL
LIN {X 0,Y 336.425,Z 1106.425,A -85,B 0,C 180,E1 21285.423,E2 21285.423} C_VEL
LIN {X 0,Y 323.269,Z 1124.456,A -85,B 0,C 180,E1 21293.418,E2 21293.418} C_VEL
LIN {X 0,Y 315.58,Z 1136.359,A -85,B 0,C 180,E1 21301.392,E2 21301.392} C_VEL
LIN {X 0,Y 311.825,Z 1143.171,A -85,B 0,C 180,E1 21308.689,E2 21308.689} C_VEL
LIN {X 0,Y 310.105,Z 1146.499,A -85,B 0,C 180,E1 21315.9,E2 21315.9} C_VEL
LIN {X 0,Y 310.127,Z 1146.137,A -85,B 0,C 180,E1 21324.409,E2 21324.409} C_VEL
LIN {X 0,Y 311.472,Z 1142.389,A -85,B 0,C 180,E1 21331.391,E2 21331.391} C_VEL
LIN {X 0,Y 314.414,Z 1134.126,A -85,B 0,C 180,E1 21339.361,E2 21339.361} C_VEL
LIN {X 0,Y 321.375,Z 1120.102,A -85,B 0,C 180,E1 21347.798,E2 21347.798} C_VEL
LIN {X 0,Y 333.936,Z 1098.96,A -85,B 0,C 180,E1 21356.182,E2 21356.182} C_VEL
LIN {X 0,Y 349.432,Z 1073.607,A -85,B 0,C 180,E1 21363.093,E2 21363.093} C_VEL
LIN {X 0,Y 366.874,Z 1043.935,A -85,B 0,C 180,E1 21368.914,E2 21368.914} C_VEL
LIN {X 0,Y 386.468,Z 1007.557,A -85,B 0,C 180,E1 21373.971,E2 21373.971} C_VEL
LIN {X 0,Y 403.759,Z 970.521,A -85,B 0,C 180,E1 21377.667,E2 21377.667} C_VEL
LIN {X 0,Y 418.66,Z 932.423,A -85,B 0,C 180,E1 21380.502,E2 21380.502} C_VEL
LIN {X 0,Y 413.276,Z 907.782,A -85,B 0,C 180,E1 21385.468,E2 21385.468} C_VEL
LIN {X 0,Y 406.964,Z 887.311,A -85,B 0,C 180,E1 21390.503,E2 21390.503} C_VEL
LIN {X 0,Y 399.842,Z 869.11,A -85,B 0,C 180,E1 21396.507,E2 21396.507} C_VEL
LIN {X 0,Y 395.475,Z 859.606,A -85,B 0,C 180,E1 21401.04,E2 21401.04} C_VEL
LIN {X 0,Y 393.391,Z 854.843,A -85,B 0,C 180,E1 21404.009,E2 21404.009} C_VEL
LIN {X 0,Y 391.867,Z 849.773,A -85,B 0,C 180,E1 21407.931,E2 21407.931} C_VEL
LIN {X 0,Y 391.764,Z 849.026,A -85,B 0,C 180,E1 21416.541,E2 21416.541} C_VEL
LIN {X 0,Y 393.396,Z 851.072,A -85,B 0,C 180,E1 21419.785,E2 21419.785} C_VEL
LIN {X 0,Y 396.955,Z 858.848,A -85,B 0,C 180,E1 21424.72,E2 21424.72} C_VEL
LIN {X 0,Y 402.533,Z 870.261,A -85,B 0,C 180,E1 21429.72,E2 21429.72} C_VEL
LIN {X 0,Y 409.951,Z 887.035,A -85,B 0,C 180,E1 21434.947,E2 21434.947} C_VEL
LIN {X 0,Y 418.214,Z 909.888,A -85,B 0,C 180,E1 21440.205,E2 21440.205} C_VEL
LIN {X 0,Y 426.011,Z 938.173,A -85,B 0,C 180,E1 21445.364,E2 21445.364} C_VEL
LIN {X 0,Y 409.444,Z 984.938,A -85,B 0,C 180,E1 21448.294,E2 21448.294} C_VEL
LIN {X 0,Y 391.933,Z 1025.402,A -85,B 0,C 180,E1 21451.751,E2 21451.751} C_VEL
LIN {X 0,Y 371.684,Z 1066.332,A -85,B 0,C 180,E1 21456.584,E2 21456.584} C_VEL
LIN {X 0,Y 352.782,Z 1101.457,A -85,B 0,C 180,E1 21462.417,E2 21462.417} C_VEL
LIN {X 0,Y 336.676,Z 1130.958,A -85,B 0,C 180,E1 21469.128,E2 21469.128} C_VEL
LIN {X 0,Y 323.363,Z 1156.521,A -85,B 0,C 180,E1 21477.252,E2 21477.252} C_VEL
LIN {X 0,Y 315.18,Z 1175.249,A -85,B 0,C 180,E1 21485.622,E2 21485.622} C_VEL
LIN {X 0,Y 311.471,Z 1186.846,A -85,B 0,C 180,E1 21493.075,E2 21493.075} C_VEL
LIN {X 0,Y 310.119,Z 1194.054,A -85,B 0,C 180,E1 21500.179,E2 21500.179} C_VEL
LIN {X 0,Y 309.966,Z 1197.573,A -85,B 0,C 180,E1 21507.204,E2 21507.204} C_VEL
LIN {X 0,Y 310.068,Z 1197.656,A -85,B 0,C 180,E1 21512.792,E2 21512.792} C_VEL
LIN {X 0,Y 310.185,Z 1193.597,A -85,B 0,C 180,E1 21521.236,E2 21521.236} C_VEL
LIN {X 0,Y 311.931,Z 1186.323,A -85,B 0,C 180,E1 21528.295,E2 21528.295} C_VEL
LIN {X 0,Y 317.208,Z 1172.756,A -85,B 0,C 180,E1 21536.907,E2 21536.907} C_VEL
LIN {X 0,Y 328.332,Z 1151.79,A -85,B 0,C 180,E1 21545.929,E2 21545.929} C_VEL
LIN {X 0,Y 343.598,Z 1126.773,A -85,B 0,C 180,E1 21553.589,E2 21553.589} C_VEL
LIN {X 0,Y 364.041,Z 1094.448,A -85,B 0,C 180,E1 21560.633,E2 21560.633} C_VEL
LIN {X 0,Y 384.8,Z 1060.276,A -85,B 0,C 180,E1 21565.931,E2 21565.931} C_VEL
LIN {X 0,Y 407.271,Z 1019.953,A -85,B 0,C 180,E1 21570.412,E2 21570.412} C_VEL
LIN {X 0,Y 426.279,Z 980.466,A -85,B 0,C 180,E1 21573.531,E2 21573.531} C_VEL
LIN {X 0,Y 440.859,Z 944.335,A -85,B 0,C 180,E1 21575.717,E2 21575.717} C_VEL
LIN {X 0,Y 436.156,Z 924.724,A -85,B 0,C 180,E1 21580.631,E2 21580.631} C_VEL
LIN {X 0,Y 434.052,Z 917.857,A -85,B 0,C 180,E1 21582.835,E2 21582.835} C_VEL
LIN {X 0,Y 431.494,Z 915.764,A -85,B 0,C 180,E1 21584.52,E2 21584.52} C_VEL
LIN {X 0,Y 427.409,Z 914.626,A -85,B 0,C 180,E1 21587.118,E2 21587.118} C_VEL
LIN {X 0,Y 427.207,Z 914.082,A -85,B 0,C 180,E1 21587.404,E2 21587.404} C_VEL
LIN {X 0,Y 424.785,Z 907.257,A -85,B 0,C 180,E1 21591.825,E2 21591.825} C_VEL
LIN {X 0,Y 423.733,Z 902.754,A -85,B 0,C 180,E1 21596.887,E2 21596.887} C_VEL
LIN {X 0,Y 423.605,Z 903.696,A -85,B 0,C 180,E1 21601.028,E2 21601.028} C_VEL
LIN {X 0,Y 424.595,Z 911.512,A -85,B 0,C 180,E1 21607.161,E2 21607.161} C_VEL
LIN {X 0,Y 427.132,Z 924.018,A -85,B 0,C 180,E1 21612.781,E2 21612.781} C_VEL
LIN {X 0,Y 429.755,Z 940.763,A -85,B 0,C 180,E1 21617.979,E2 21617.979} C_VEL
LIN {X 0,Y 430.284,Z 947.886,A -85,B 0,C 180,E1 21619.689,E2 21619.689} C_VEL
LIN {X 0,Y 410.062,Z 989.163,A -85,B 0,C 180,E1 21622.889,E2 21622.889} C_VEL
LIN {X 0,Y 389.875,Z 1023.864,A -85,B 0,C 180,E1 21626.608,E2 21626.608} C_VEL
LIN {X 0,Y 366.615,Z 1058.71,A -85,B 0,C 180,E1 21631.946,E2 21631.946} C_VEL
LIN {X 0,Y 345.865,Z 1086.715,A -85,B 0,C 180,E1 21638.148,E2 21638.148} C_VEL
LIN {X 0,Y 328.739,Z 1109.01,A -85,B 0,C 180,E1 21645.215,E2 21645.215} C_VEL
LIN {X 0,Y 314.68,Z 1127.43,A -85,B 0,C 180,E1 21653.968,E2 21653.968} C_VEL
LIN {X 0,Y 307.013,Z 1138.812,A -85,B 0,C 180,E1 21662.39,E2 21662.39} C_VEL
LIN {X 0,Y 303.597,Z 1144.685,A -85,B 0,C 180,E1 21669.611,E2 21669.611} C_VEL
LIN {X 0,Y 301.969,Z 1147.504,A -85,B 0,C 180,E1 21678.455,E2 21678.455} C_VEL
LIN {X 0,Y 302.702,Z 1145.805,A -85,B 0,C 180,E1 21687.14,E2 21687.14} C_VEL
LIN {X 0,Y 304.277,Z 1140.903,A -85,B 0,C 180,E1 21694.274,E2 21694.274} C_VEL
LIN {X 0,Y 308.839,Z 1130.604,A -85,B 0,C 180,E1 21702.721,E2 21702.721} C_VEL
LIN {X 0,Y 317.387,Z 1115.362,A -85,B 0,C 180,E1 21710.923,E2 21710.923} C_VEL
LIN {X 0,Y 330.681,Z 1094.049,A -85,B 0,C 180,E1 21718.675,E2 21718.675} C_VEL
LIN {X 0,Y 346.931,Z 1068.517,A -85,B 0,C 180,E1 21725.251,E2 21725.251} C_VEL
LIN {X 0,Y 366.663,Z 1035.413,A -85,B 0,C 180,E1 21731.256,E2 21731.256} C_VEL
LIN {X 0,Y 385.109,Z 1000.797,A -85,B 0,C 180,E1 21735.736,E2 21735.736} C_VEL
LIN {X 0,Y 403.266,Z 961.889,A -85,B 0,C 180,E1 21739.361,E2 21739.361} C_VEL
LIN {X 0,Y 413.139,Z 936.739,A -85,B 0,C 180,E1 21741.162,E2 21741.162} C_VEL
LIN {X 0,Y 409.366,Z 915.581,A -85,B 0,C 180,E1 21745.447,E2 21745.447} C_VEL
LIN {X 0,Y 403.999,Z 895.882,A -85,B 0,C 180,E1 21750.282,E2 21750.282} C_VEL
LIN {X 0,Y 397.181,Z 877.05,A -85,B 0,C 180,E1 21756.446,E2 21756.446} C_VEL
LIN {X 0,Y 393.2,Z 867.445,A -85,B 0,C 180,E1 21760.926,E2 21760.926} C_VEL
LIN {X 0,Y 390.893,Z 862.02,A -85,B 0,C 180,E1 21764.436,E2 21764.436} C_VEL
LIN {X 0,Y 389.521,Z 857.204,A -85,B 0,C 180,E1 21768.334,E2 21768.334} C_VEL
LIN {X 0,Y 389.726,Z 856.696,A -85,B 0,C 180,E1 21776.659,E2 21776.659} C_VEL
LIN {X 0,Y 391.185,Z 858.728,A -85,B 0,C 180,E1 21779.714,E2 21779.714} C_VEL
LIN {X 0,Y 394.616,Z 866.488,A -85,B 0,C 180,E1 21784.657,E2 21784.657} C_VEL
LIN {X 0,Y 400.521,Z 879.042,A -85,B 0,C 180,E1 21790.112,E2 21790.112} C_VEL
LIN {X 0,Y 408.257,Z 898.502,A -85,B 0,C 180,E1 21795.842,E2 21795.842} C_VEL
LIN {X 0,Y 415.625,Z 921.55,A -85,B 0,C 180,E1 21800.949,E2 21800.949} C_VEL
LIN {X 0,Y 420.436,Z 942.691,A -85,B 0,C 180,E1 21804.74,E2 21804.74} C_VEL
LIN {X 0,Y 403.833,Z 987.357,A -85,B 0,C 180,E1 21807.549,E2 21807.549} C_VEL
LIN {X 0,Y 385.341,Z 1028.481,A -85,B 0,C 180,E1 21811.164,E2 21811.164} C_VEL
LIN {X 0,Y 365.585,Z 1067.101,A -85,B 0,C 180,E1 21815.811,E2 21815.811} C_VEL
LIN {X 0,Y 345.478,Z 1103.227,A -85,B 0,C 180,E1 21821.961,E2 21821.961} C_VEL
LIN {X 0,Y 329.094,Z 1132.031,A -85,B 0,C 180,E1 21828.761,E2 21828.761} C_VEL
LIN {X 0,Y 315.295,Z 1157.754,A -85,B 0,C 180,E1 21837.248,E2 21837.248} C_VEL
LIN {X 0,Y 307.075,Z 1175.959,A -85,B 0,C 180,E1 21845.878,E2 21845.878} C_VEL
LIN {X 0,Y 303.271,Z 1187.806,A -85,B 0,C 180,E1 21854.093,E2 21854.093} C_VEL
LIN {X 0,Y 302.111,Z 1194.293,A -85,B 0,C 180,E1 21861.368,E2 21861.368} C_VEL
LIN {X 0,Y 302.21,Z 1197.192,A -85,B 0,C 180,E1 21869.355,E2 21869.355} C_VEL
LIN {X 0,Y 301.951,Z 1196.218,A -85,B 0,C 180,E1 21875.743,E2 21875.743} C_VEL
LIN {X 0,Y 302.63,Z 1191.423,A -85,B 0,C 180,E1 21883.38,E2 21883.38} C_VEL
LIN {X 0,Y 305.644,Z 1181.713,A -85,B 0,C 180,E1 21891.764,E2 21891.764} C_VEL
LIN {X 0,Y 312.735,Z 1166.477,A -85,B 0,C 180,E1 21900.485,E2 21900.485} C_VEL
LIN {X 0,Y 325.118,Z 1145.477,A -85,B 0,C 180,E1 21908.862,E2 21908.862} C_VEL
LIN {X 0,Y 343.596,Z 1117.236,A -85,B 0,C 180,E1 21916.854,E2 21916.854} C_VEL
LIN {X 0,Y 364.553,Z 1085.163,A -85,B 0,C 180,E1 21923.208,E2 21923.208} C_VEL
LIN {X 0,Y 386.528,Z 1049.682,A -85,B 0,C 180,E1 21928.264,E2 21928.264} C_VEL
LIN {X 0,Y 409.116,Z 1008.39,A -85,B 0,C 180,E1 21932.431,E2 21932.431} C_VEL
LIN {X 0,Y 429.28,Z 965.596,A -85,B 0,C 180,E1 21935.459,E2 21935.459} C_VEL
LIN {X 0,Y 436.1,Z 948.481,A -85,B 0,C 180,E1 21936.469,E2 21936.469} C_VEL
LIN {X 0,Y 432.195,Z 930.649,A -85,B 0,C 180,E1 21941.108,E2 21941.108} C_VEL
LIN {X 0,Y 427.975,Z 916.654,A -85,B 0,C 180,E1 21946.217,E2 21946.217} C_VEL
LIN {X 0,Y 427.207,Z 914.082,A -85,B 0,C 180,E1 21947.404,E2 21947.404} C_VEL
LIN {X 0,Y 425.177,Z 913.148,A -85,B 0,C 180,E1 21949.14,E2 21949.14} C_VEL
LIN {X 0,Y 421.49,Z 914.251,A -85,B 0,C 180,E1 21952.1,E2 21952.1} C_VEL
LIN {X 0,Y 420.85,Z 910.38,A -85,B 0,C 180,E1 21955.887,E2 21955.887} C_VEL
LIN {X 0,Y 420.572,Z 910.069,A -85,B 0,C 180,E1 21960.006,E2 21960.006} C_VEL
LIN {X 0,Y 421.029,Z 917.168,A -85,B 0,C 180,E1 21966.187,E2 21966.187} C_VEL
LIN {X 0,Y 422.932,Z 928.942,A -85,B 0,C 180,E1 21971.862,E2 21971.862} C_VEL
LIN {X 0,Y 425.082,Z 944.725,A -85,B 0,C 180,E1 21977.061,E2 21977.061} C_VEL
LIN {X 0,Y 425.502,Z 952.019,A -85,B 0,C 180,E1 21978.947,E2 21978.947} C_VEL
LIN {X 0,Y 404.909,Z 992.691,A -85,B 0,C 180,E1 21982.143,E2 21982.143} C_VEL
LIN {X 0,Y 384.221,Z 1026.853,A -85,B 0,C 180,E1 21985.888,E2 21985.888} C_VEL
LIN {X 0,Y 360.96,Z 1060.612,A -85,B 0,C 180,E1 21991.135,E2 21991.135} C_VEL
LIN {X 0,Y 339.786,Z 1088.071,A -85,B 0,C 180,E1 21997.323,E2 21997.323} C_VEL
LIN {X 0,Y 322.301,Z 1109.875,A -85,B 0,C 180,E1 22004.36,E2 22004.36} C_VEL
LIN {X 0,Y 307.74,Z 1128.007,A -85,B 0,C 180,E1 22013.13,E2 22013.13} C_VEL
LIN {X 0,Y 299.617,Z 1139.336,A -85,B 0,C 180,E1 22021.648,E2 22021.648} C_VEL
LIN {X 0,Y 295.922,Z 1145.268,A -85,B 0,C 180,E1 22029.058,E2 22029.058} C_VEL
LIN {X 0,Y 294.119,Z 1148.143,A -85,B 0,C 180,E1 22038.142,E2 22038.142} C_VEL
LIN {X 0,Y 294.783,Z 1146.528,A -85,B 0,C 180,E1 22047.063,E2 22047.063} C_VEL
LIN {X 0,Y 296.441,Z 1141.695,A -85,B 0,C 180,E1 22054.387,E2 22054.387} C_VEL
LIN {X 0,Y 301.194,Z 1131.494,A -85,B 0,C 180,E1 22063.05,E2 22063.05} C_VEL
LIN {X 0,Y 311.016,Z 1114.822,A -85,B 0,C 180,E1 22072.122,E2 22072.122} C_VEL
LIN {X 0,Y 326.603,Z 1091.097,A -85,B 0,C 180,E1 22080.595,E2 22080.595} C_VEL
LIN {X 0,Y 344.012,Z 1064.31,A -85,B 0,C 180,E1 22087.158,E2 22087.158} C_VEL
LIN {X 0,Y 362.937,Z 1033.445,A -85,B 0,C 180,E1 22092.579,E2 22092.579} C_VEL
LIN {X 0,Y 383.154,Z 995.906,A -85,B 0,C 180,E1 22097.271,E2 22097.271} C_VEL
LIN {X 0,Y 401.266,Z 956.714,A -85,B 0,C 180,E1 22100.749,E2 22100.749} C_VEL
LIN {X 0,Y 408.029,Z 939.526,A -85,B 0,C 180,E1 22101.994,E2 22101.994} C_VEL
LIN {X 0,Y 403.663,Z 915.979,A -85,B 0,C 180,E1 22107.117,E2 22107.117} C_VEL
LIN {X 0,Y 398.341,Z 896.572,A -85,B 0,C 180,E1 22112.349,E2 22112.349} C_VEL
LIN {X 0,Y 392.906,Z 880.809,A -85,B 0,C 180,E1 22118.087,E2 22118.087} C_VEL
LIN {X 0,Y 389.355,Z 871.107,A -85,B 0,C 180,E1 22123.07,E2 22123.07} C_VEL
LIN {X 0,Y 387.389,Z 864.857,A -85,B 0,C 180,E1 22128.176,E2 22128.176} C_VEL
LIN {X 0,Y 387.53,Z 864.274,A -85,B 0,C 180,E1 22136.641,E2 22136.641} C_VEL
LIN {X 0,Y 388.881,Z 866.278,A -85,B 0,C 180,E1 22139.576,E2 22139.576} C_VEL
LIN {X 0,Y 392.084,Z 873.756,A -85,B 0,C 180,E1 22144.415,E2 22144.415} C_VEL
LIN {X 0,Y 397.84,Z 887.055,A -85,B 0,C 180,E1 22150.181,E2 22150.181} C_VEL
LIN {X 0,Y 404.754,Z 905.877,A -85,B 0,C 180,E1 22155.711,E2 22155.711} C_VEL
LIN {X 0,Y 411.371,Z 928.137,A -85,B 0,C 180,E1 22160.7,E2 22160.7} C_VEL
LIN {X 0,Y 415.247,Z 945.582,A -85,B 0,C 180,E1 22163.961,E2 22163.961} C_VEL
LIN {X 0,Y 398.392,Z 989.385,A -85,B 0,C 180,E1 22166.767,E2 22166.767} C_VEL
LIN {X 0,Y 378.583,Z 1032.021,A -85,B 0,C 180,E1 22170.607,E2 22170.607} C_VEL
LIN {X 0,Y 359.358,Z 1068.137,A -85,B 0,C 180,E1 22175.069,E2 22175.069} C_VEL
LIN {X 0,Y 338.631,Z 1104.202,A -85,B 0,C 180,E1 22181.324,E2 22181.324} C_VEL
LIN {X 0,Y 321.508,Z 1133.176,A -85,B 0,C 180,E1 22188.401,E2 22188.401} C_VEL
LIN {X 0,Y 308.202,Z 1156.941,A -85,B 0,C 180,E1 22196.45,E2 22196.45} C_VEL
LIN {X 0,Y 299.57,Z 1175.096,A -85,B 0,C 180,E1 22205.211,E2 22205.211} C_VEL
LIN {X 0,Y 295.5,Z 1187.046,A -85,B 0,C 180,E1 22213.663,E2 22213.663} C_VEL
LIN {X 0,Y 294.241,Z 1193.589,A -85,B 0,C 180,E1 22221.136,E2 22221.136} C_VEL
LIN {X 0,Y 294.195,Z 1196.253,A -85,B 0,C 180,E1 22227.054,E2 22227.054} C_VEL
LIN {X 0,Y 294.288,Z 1196.368,A -85,B 0,C 180,E1 22232.942,E2 22232.942} C_VEL
LIN {X 0,Y 294.149,Z 1194.31,A -85,B 0,C 180,E1 22238.864,E2 22238.864} C_VEL
LIN {X 0,Y 295.425,Z 1188.471,A -85,B 0,C 180,E1 22246.338,E2 22246.338} C_VEL
LIN {X 0,Y 299.597,Z 1177.582,A -85,B 0,C 180,E1 22254.8,E2 22254.8} C_VEL
LIN {X 0,Y 309.902,Z 1158.699,A -85,B 0,C 180,E1 22264.563,E2 22264.563} C_VEL
LIN {X 0,Y 324.908,Z 1135.576,A -85,B 0,C 180,E1 22272.856,E2 22272.856} C_VEL
LIN {X 0,Y 345.9,Z 1105.158,A -85,B 0,C 180,E1 22280.494,E2 22280.494} C_VEL
LIN {X 0,Y 368.51,Z 1071.17,A -85,B 0,C 180,E1 22286.431,E2 22286.431} C_VEL
LIN {X 0,Y 391.558,Z 1033.77,A -85,B 0,C 180,E1 22291.054,E2 22291.054} C_VEL
LIN {X 0,Y 413.019,Z 993.496,A -85,B 0,C 180,E1 22294.586,E2 22294.586} C_VEL
LIN {X 0,Y 430.803,Z 954.176,A -85,B 0,C 180,E1 22297.101,E2 22297.101} C_VEL
LIN {X 0,Y 430.686,Z 949.022,A -85,B 0,C 180,E1 22298.117,E2 22298.117} C_VEL
LIN {X 0,Y 426.833,Z 931.786,A -85,B 0,C 180,E1 22303.17,E2 22303.17} C_VEL
LIN {X 0,Y 423.133,Z 919.045,A -85,B 0,C 180,E1 22308.678,E2 22308.678} C_VEL
LIN {X 0,Y 421.49,Z 914.251,A -85,B 0,C 180,E1 22312.1,E2 22312.1} C_VEL
LIN {X 0,Y 419.315,Z 915.349,A -85,B 0,C 180,E1 22314.455,E2 22314.455} C_VEL
LIN {X 0,Y 417.467,Z 917.378,A -85,B 0,C 180,E1 22316.843,E2 22316.843} C_VEL
LIN {X 0,Y 417.353,Z 917.355,A -85,B 0,C 180,E1 22320.006,E2 22320.006} C_VEL
LIN {X 0,Y 417.564,Z 924.485,A -85,B 0,C 180,E1 22326.239,E2 22326.239} C_VEL
LIN {X 0,Y 419.188,Z 936.439,A -85,B 0,C 180,E1 22331.969,E2 22331.969} C_VEL
LIN {X 0,Y 420.742,Z 952.412,A -85,B 0,C 180,E1 22337.207,E2 22337.207} C_VEL
LIN {X 0,Y 420.517,Z 956.69,A -85,B 0,C 180,E1 22338.22,E2 22338.22} C_VEL
LIN {X 0,Y 399.497,Z 996.666,A -85,B 0,C 180,E1 22341.423,E2 22341.423} C_VEL
LIN {X 0,Y 376.601,Z 1032.901,A -85,B 0,C 180,E1 22345.561,E2 22345.561} C_VEL
LIN {X 0,Y 354.631,Z 1063.364,A -85,B 0,C 180,E1 22350.483,E2 22350.483} C_VEL
LIN {X 0,Y 331.805,Z 1091.923,A -85,B 0,C 180,E1 22357.158,E2 22357.158} C_VEL
LIN {X 0,Y 313.396,Z 1113.618,A -85,B 0,C 180,E1 22364.681,E2 22364.681} C_VEL
LIN {X 0,Y 300.138,Z 1129.551,A -85,B 0,C 180,E1 22372.832,E2 22372.832} C_VEL
LIN {X 0,Y 291.38,Z 1141.058,A -85,B 0,C 180,E1 22382.178,E2 22382.178} C_VEL
LIN {X 0,Y 287.295,Z 1147.214,A -85,B 0,C 180,E1 22391.252,E2 22391.252} C_VEL
LIN {X 0,Y 286.279,Z 1148.784,A -85,B 0,C 180,E1 22397.812,E2 22397.812} C_VEL
LIN {X 0,Y 286.891,Z 1147.23,A -85,B 0,C 180,E1 22406.982,E2 22406.982} C_VEL
LIN {X 0,Y 288.614,Z 1142.465,A -85,B 0,C 180,E1 22414.506,E2 22414.506} C_VEL
LIN {X 0,Y 293.547,Z 1132.383,A -85,B 0,C 180,E1 22423.396,E2 22423.396} C_VEL
LIN {X 0,Y 303.784,Z 1115.84,A -85,B 0,C 180,E1 22432.677,E2 22432.677} C_VEL
LIN {X 0,Y 319.159,Z 1093.224,A -85,B 0,C 180,E1 22440.992,E2 22440.992} C_VEL
LIN {X 0,Y 336.939,Z 1066.962,A -85,B 0,C 180,E1 22447.668,E2 22447.668} C_VEL
LIN {X 0,Y 357.26,Z 1034.905,A -85,B 0,C 180,E1 22453.421,E2 22453.421} C_VEL
LIN {X 0,Y 377.362,Z 998.669,A -85,B 0,C 180,E1 22458.017,E2 22458.017} C_VEL
LIN {X 0,Y 395.871,Z 960.197,A -85,B 0,C 180,E1 22461.495,E2 22461.495} C_VEL
LIN {X 0,Y 402.729,Z 943.677,A -85,B 0,C 180,E1 22462.693,E2 22462.693} C_VEL
LIN {X 0,Y 399.171,Z 921.562,A -85,B 0,C 180,E1 22467.588,E2 22467.588} C_VEL
LIN {X 0,Y 394.619,Z 903.26,A -85,B 0,C 180,E1 22472.636,E2 22472.636} C_VEL
LIN {X 0,Y 389.557,Z 887.303,A -85,B 0,C 180,E1 22478.592,E2 22478.592} C_VEL
LIN {X 0,Y 386.147,Z 877.496,A -85,B 0,C 180,E1 22484.095,E2 22484.095} C_VEL
LIN {X 0,Y 384.795,Z 872.251,A -85,B 0,C 180,E1 22488.669,E2 22488.669} C_VEL
LIN {X 0,Y 384.877,Z 871.508,A -85,B 0,C 180,E1 22495.49,E2 22495.49} C_VEL
LIN {X 0,Y 386.349,Z 872.811,A -85,B 0,C 180,E1 22498.873,E2 22498.873} C_VEL
LIN {X 0,Y 390.477,Z 883.332,A -85,B 0,C 180,E1 22505.546,E2 22505.546} C_VEL
LIN {X 0,Y 396.468,Z 898.888,A -85,B 0,C 180,E1 22511.537,E2 22511.537} C_VEL
LIN {X 0,Y 403.139,Z 919.598,A -85,B 0,C 180,E1 22517.163,E2 22517.163} C_VEL
LIN {X 0,Y 409.042,Z 944.116,A -85,B 0,C 180,E1 22522.302,E2 22522.302} C_VEL
LIN {X 0,Y 409.582,Z 950.091,A -85,B 0,C 180,E1 22523.255,E2 22523.255} C_VEL
LIN {X 0,Y 392.143,Z 993.252,A -85,B 0,C 180,E1 22526.115,E2 22526.115} C_VEL
LIN {X 0,Y 372.512,Z 1034.185,A -85,B 0,C 180,E1 22529.883,E2 22529.883} C_VEL
LIN {X 0,Y 352.032,Z 1071.085,A -85,B 0,C 180,E1 22534.583,E2 22534.583} C_VEL
LIN {X 0,Y 332.023,Z 1104.822,A -85,B 0,C 180,E1 22540.588,E2 22540.588} C_VEL
LIN {X 0,Y 313.72,Z 1134.661,A -85,B 0,C 180,E1 22548.125,E2 22548.125} C_VEL
LIN {X 0,Y 300.194,Z 1157.958,A -85,B 0,C 180,E1 22556.376,E2 22556.376} C_VEL
LIN {X 0,Y 291.429,Z 1175.832,A -85,B 0,C 180,E1 22565.49,E2 22565.49} C_VEL
LIN {X 0,Y 287.749,Z 1186.286,A -85,B 0,C 180,E1 22573.21,E2 22573.21} C_VEL
LIN {X 0,Y 286.371,Z 1192.883,A -85,B 0,C 180,E1 22580.89,E2 22580.89} C_VEL
LIN {X 0,Y 286.302,Z 1195.591,A -85,B 0,C 180,E1 22586.973,E2 22586.973} C_VEL
LIN {X 0,Y 286.416,Z 1195.725,A -85,B 0,C 180,E1 22593.023,E2 22593.023} C_VEL
LIN {X 0,Y 286.258,Z 1193.695,A -85,B 0,C 180,E1 22599.111,E2 22599.111} C_VEL
LIN {X 0,Y 287.647,Z 1187.865,A -85,B 0,C 180,E1 22606.793,E2 22606.793} C_VEL
LIN {X 0,Y 292.121,Z 1177.024,A -85,B 0,C 180,E1 22615.479,E2 22615.479} C_VEL
LIN {X 0,Y 303.237,Z 1157.989,A -85,B 0,C 180,E1 22625.54,E2 22625.54} C_VEL
LIN {X 0,Y 318.848,Z 1135.129,A -85,B 0,C 180,E1 22633.876,E2 22633.876} C_VEL
LIN {X 0,Y 340.958,Z 1104.391,A -85,B 0,C 180,E1 22641.657,E2 22641.657} C_VEL
LIN {X 0,Y 363.941,Z 1070.984,A -85,B 0,C 180,E1 22647.5,E2 22647.5} C_VEL
LIN {X 0,Y 387.635,Z 1033.611,A -85,B 0,C 180,E1 22652.115,E2 22652.115} C_VEL
LIN {X 0,Y 409.609,Z 993.423,A -85,B 0,C 180,E1 22655.609,E2 22655.609} C_VEL
LIN {X 0,Y 426.382,Z 957.388,A -85,B 0,C 180,E1 22657.915,E2 22657.915} C_VEL
LIN {X 0,Y 423.912,Z 942.561,A -85,B 0,C 180,E1 22661.98,E2 22661.98} C_VEL
LIN {X 0,Y 420.455,Z 928.52,A -85,B 0,C 180,E1 22667.552,E2 22667.552} C_VEL
LIN {X 0,Y 418.037,Z 920.824,A -85,B 0,C 180,E1 22672.737,E2 22672.737} C_VEL
LIN {X 0,Y 417.467,Z 917.378,A -85,B 0,C 180,E1 22676.843,E2 22676.843} C_VEL
LIN {X 0,Y 416.319,Z 919.492,A -85,B 0,C 180,E1 22678.616,E2 22678.616} C_VEL
LIN {X 0,Y 413.674,Z 926.132,A -85,B 0,C 180,E1 22681.537,E2 22681.537} C_VEL
LIN {X 0,Y 413.965,Z 931.779,A -85,B 0,C 180,E1 22686.293,E2 22686.293} C_VEL
LIN {X 0,Y 415.168,Z 943.862,A -85,B 0,C 180,E1 22692.087,E2 22692.087} C_VEL
LIN {X 0,Y 416.186,Z 959.847,A -85,B 0,C 180,E1 22697.311,E2 22697.311} C_VEL
LIN {X 0,Y 395.046,Z 998.991,A -85,B 0,C 180,E1 22700.538,E2 22700.538} C_VEL
LIN {X 0,Y 371.362,Z 1035.407,A -85,B 0,C 180,E1 22704.732,E2 22704.732} C_VEL
LIN {X 0,Y 348.312,Z 1066.128,A -85,B 0,C 180,E1 22709.812,E2 22709.812} C_VEL
LIN {X 0,Y 325.602,Z 1093.559,A -85,B 0,C 180,E1 22716.36,E2 22716.36} C_VEL
LIN {X 0,Y 305.356,Z 1116.367,A -85,B 0,C 180,E1 22724.588,E2 22724.588} C_VEL
LIN {X 0,Y 291.842,Z 1131.861,A -85,B 0,C 180,E1 22733.093,E2 22733.093} C_VEL
LIN {X 0,Y 282.976,Z 1143.024,A -85,B 0,C 180,E1 22743.007,E2 22743.007} C_VEL
LIN {X 0,Y 279.491,Z 1147.964,A -85,B 0,C 180,E1 22751.072,E2 22751.072} C_VEL
LIN {X 0,Y 278.285,Z 1149.436,A -85,B 0,C 180,E1 22760.626,E2 22760.626} C_VEL
LIN {X 0,Y 278.981,Z 1147.933,A -85,B 0,C 180,E1 22766.897,E2 22766.897} C_VEL
LIN {X 0,Y 280.795,Z 1143.234,A -85,B 0,C 180,E1 22774.632,E2 22774.632} C_VEL
LIN {X 0,Y 285.904,Z 1133.273,A -85,B 0,C 180,E1 22783.761,E2 22783.761} C_VEL
LIN {X 0,Y 296.589,Z 1116.789,A -85,B 0,C 180,E1 22793.287,E2 22793.287} C_VEL
LIN {X 0,Y 312.475,Z 1094.335,A -85,B 0,C 180,E1 22801.731,E2 22801.731} C_VEL
LIN {X 0,Y 330.802,Z 1068.236,A -85,B 0,C 180,E1 22808.493,E2 22808.493} C_VEL
LIN {X 0,Y 351.498,Z 1036.554,A -85,B 0,C 180,E1 22814.254,E2 22814.254} C_VEL
LIN {X 0,Y 371.642,Z 1001.425,A -85,B 0,C 180,E1 22818.785,E2 22818.785} C_VEL
LIN {X 0,Y 391.146,Z 962.228,A -85,B 0,C 180,E1 22822.373,E2 22822.373} C_VEL
LIN {X 0,Y 397.552,Z 946.318,A -85,B 0,C 180,E1 22823.653,E2 22823.653} C_VEL
LIN {X 0,Y 394.201,Z 924.426,A -85,B 0,C 180,E1 22828.75,E2 22828.75} C_VEL
LIN {X 0,Y 390.345,Z 907.932,A -85,B 0,C 180,E1 22833.555,E2 22833.555} C_VEL
LIN {X 0,Y 386.006,Z 893.211,A -85,B 0,C 180,E1 22839.363,E2 22839.363} C_VEL
LIN {X 0,Y 383.04,Z 883.897,A -85,B 0,C 180,E1 22845.135,E2 22845.135} C_VEL
LIN {X 0,Y 382.291,Z 879.753,A -85,B 0,C 180,E1 22848.594,E2 22848.594} C_VEL
LIN {X 0,Y 382.34,Z 878.985,A -85,B 0,C 180,E1 22855.46,E2 22855.46} C_VEL
LIN {X 0,Y 383.826,Z 881.047,A -85,B 0,C 180,E1 22859.228,E2 22859.228} C_VEL
LIN {X 0,Y 387.818,Z 891.188,A -85,B 0,C 180,E1 22865.584,E2 22865.584} C_VEL
LIN {X 0,Y 393.397,Z 906.898,A -85,B 0,C 180,E1 22871.628,E2 22871.628} C_VEL
LIN {X 0,Y 399.555,Z 927.88,A -85,B 0,C 180,E1 22877.297,E2 22877.297} C_VEL
LIN {X 0,Y 404.646,Z 951.612,A -85,B 0,C 180,E1 22882.272,E2 22882.272} C_VEL
LIN {X 0,Y 386.609,Z 995.642,A -85,B 0,C 180,E1 22885.325,E2 22885.325} C_VEL
LIN {X 0,Y 366.38,Z 1036.484,A -85,B 0,C 180,E1 22889.156,E2 22889.156} C_VEL
LIN {X 0,Y 344.35,Z 1074.817,A -85,B 0,C 180,E1 22894.212,E2 22894.212} C_VEL
LIN {X 0,Y 324.351,Z 1107.159,A -85,B 0,C 180,E1 22900.23,E2 22900.23} C_VEL
LIN {X 0,Y 305.155,Z 1137.403,A -85,B 0,C 180,E1 22908.217,E2 22908.217} C_VEL
LIN {X 0,Y 291.206,Z 1160.497,A -85,B 0,C 180,E1 22917.041,E2 22917.041} C_VEL
LIN {X 0,Y 282.89,Z 1177.512,A -85,B 0,C 180,E1 22926.381,E2 22926.381} C_VEL
LIN {X 0,Y 279.515,Z 1187.232,A -85,B 0,C 180,E1 22934.316,E2 22934.316} C_VEL
LIN {X 0,Y 278.502,Z 1192.176,A -85,B 0,C 180,E1 22940.63,E2 22940.63} C_VEL
LIN {X 0,Y 278.41,Z 1194.922,A -85,B 0,C 180,E1 22946.887,E2 22946.887} C_VEL
LIN {X 0,Y 278.515,Z 1195.081,A -85,B 0,C 180,E1 22953.109,E2 22953.109} C_VEL
LIN {X 0,Y 278.372,Z 1193.081,A -85,B 0,C 180,E1 22959.371,E2 22959.371} C_VEL
LIN {X 0,Y 279.894,Z 1187.259,A -85,B 0,C 180,E1 22967.272,E2 22967.272} C_VEL
LIN {X 0,Y 285.157,Z 1175.563,A -85,B 0,C 180,E1 22976.768,E2 22976.768} C_VEL
LIN {X 0,Y 296.903,Z 1156.923,A -85,B 0,C 180,E1 22986.726,E2 22986.726} C_VEL
LIN {X 0,Y 313.711,Z 1133.561,A -85,B 0,C 180,E1 22995.274,E2 22995.274} C_VEL
LIN {X 0,Y 335.871,Z 1104.014,A -85,B 0,C 180,E1 23002.767,E2 23002.767} C_VEL
LIN {X 0,Y 359.789,Z 1070.395,A -85,B 0,C 180,E1 23008.654,E2 23008.654} C_VEL
LIN {X 0,Y 384.458,Z 1032.431,A -85,B 0,C 180,E1 23013.3,E2 23013.3} C_VEL
LIN {X 0,Y 407.062,Z 991.967,A -85,B 0,C 180,E1 23016.747,E2 23016.747} C_VEL
LIN {X 0,Y 421.683,Z 961.431,A -85,B 0,C 180,E1 23018.703,E2 23018.703} C_VEL
LIN {X 0,Y 419.24,Z 946.158,A -85,B 0,C 180,E1 23023.246,E2 23023.246} C_VEL
LIN {X 0,Y 416.349,Z 933.913,A -85,B 0,C 180,E1 23028.504,E2 23028.504} C_VEL
LIN {X 0,Y 414.424,Z 926.244,A -85,B 0,C 180,E1 23034.451,E2 23034.451} C_VEL
LIN {X 0,Y 414.201,Z 924.271,A -85,B 0,C 180,E1 23037.915,E2 23037.915} C_VEL
LIN {X 0,Y 413.784,Z 925.6,A -85,B 0,C 180,E1 23041.052,E2 23041.052} C_VEL
LIN {X 0,Y 413.674,Z 926.132,A -85,B 0,C 180,E1 23041.537,E2 23041.537} C_VEL
LIN {X 0,Y 411.887,Z 932.034,A -85,B 0,C 180,E1 23043.814,E2 23043.814} C_VEL
LIN {X 0,Y 410.281,Z 938.609,A -85,B 0,C 180,E1 23046.092,E2 23046.092} C_VEL
LIN {X 0,Y 411.003,Z 949.955,A -85,B 0,C 180,E1 23051.673,E2 23051.673} C_VEL
LIN {X 0,Y 411.524,Z 964.076,A -85,B 0,C 180,E1 23056.489,E2 23056.489} C_VEL
LIN {X 0,Y 389.645,Z 1002.963,A -85,B 0,C 180,E1 23059.79,E2 23059.79} C_VEL
LIN {X 0,Y 365.522,Z 1038.859,A -85,B 0,C 180,E1 23064.019,E2 23064.019} C_VEL
LIN {X 0,Y 340.311,Z 1070.98,A -85,B 0,C 180,E1 23069.53,E2 23069.53} C_VEL
LIN {X 0,Y 317.814,Z 1096.856,A -85,B 0,C 180,E1 23076.071,E2 23076.071} C_VEL
LIN {X 0,Y 298.162,Z 1118.154,A -85,B 0,C 180,E1 23084.063,E2 23084.063} C_VEL
LIN {X 0,Y 283.951,Z 1133.555,A -85,B 0,C 180,E1 23092.981,E2 23092.981} C_VEL
LIN {X 0,Y 275.423,Z 1143.764,A -85,B 0,C 180,E1 23102.47,E2 23102.47} C_VEL
LIN {X 0,Y 271.635,Z 1148.801,A -85,B 0,C 180,E1 23111.067,E2 23111.067} C_VEL
LIN {X 0,Y 270.399,Z 1150.112,A -85,B 0,C 180,E1 23120.35,E2 23120.35} C_VEL
LIN {X 0,Y 271.095,Z 1148.633,A -85,B 0,C 180,E1 23126.806,E2 23126.806} C_VEL
LIN {X 0,Y 272.933,Z 1144.114,A -85,B 0,C 180,E1 23134.606,E2 23134.606} C_VEL
LIN {X 0,Y 278.301,Z 1134.155,A -85,B 0,C 180,E1 23144.145,E2 23144.145} C_VEL
LIN {X 0,Y 289.401,Z 1117.764,A -85,B 0,C 180,E1 23153.901,E2 23153.901} C_VEL
LIN {X 0,Y 305.833,Z 1095.439,A -85,B 0,C 180,E1 23162.504,E2 23162.504} C_VEL
LIN {X 0,Y 324.73,Z 1069.512,A -85,B 0,C 180,E1 23169.35,E2 23169.35} C_VEL
LIN {X 0,Y 346.111,Z 1037.75,A -85,B 0,C 180,E1 23175.183,E2 23175.183} C_VEL
LIN {X 0,Y 367.213,Z 1001.986,A -85,B 0,C 180,E1 23179.808,E2 23179.808} C_VEL
LIN {X 0,Y 387.138,Z 962.781,A -85,B 0,C 180,E1 23183.383,E2 23183.383} C_VEL
LIN {X 0,Y 392.286,Z 951.018,A -85,B 0,C 180,E1 23184.242,E2 23184.242} C_VEL
LIN {X 0,Y 389.92,Z 930.773,A -85,B 0,C 180,E1 23189.061,E2 23189.061} C_VEL
LIN {X 0,Y 386.085,Z 912.817,A -85,B 0,C 180,E1 23194.491,E2 23194.491} C_VEL
LIN {X 0,Y 382.585,Z 899.39,A -85,B 0,C 180,E1 23200.031,E2 23200.031} C_VEL
LIN {X 0,Y 379.895,Z 890.057,A -85,B 0,C 180,E1 23206.185,E2 23206.185} C_VEL
LIN {X 0,Y 379.683,Z 887.351,A -85,B 0,C 180,E1 23208.515,E2 23208.515} C_VEL
LIN {X 0,Y 379.802,Z 886.466,A -85,B 0,C 180,E1 23215.429,E2 23215.429} C_VEL
LIN {X 0,Y 381.233,Z 888.669,A -85,B 0,C 180,E1 23219.223,E2 23219.223} C_VEL
LIN {X 0,Y 384.715,Z 898.416,A -85,B 0,C 180,E1 23225.418,E2 23225.418} C_VEL
LIN {X 0,Y 389.697,Z 913.188,A -85,B 0,C 180,E1 23231.174,E2 23231.174} C_VEL
LIN {X 0,Y 395.307,Z 934.144,A -85,B 0,C 180,E1 23236.948,E2 23236.948} C_VEL
LIN {X 0,Y 399.222,Z 956.335,A -85,B 0,C 180,E1 23241.654,E2 23241.654} C_VEL
LIN {X 0,Y 378.965,Z 1002.68,A -85,B 0,C 180,E1 23244.876,E2 23244.876} C_VEL
LIN {X 0,Y 357.221,Z 1044.008,A -85,B 0,C 180,E1 23249.024,E2 23249.024} C_VEL
LIN {X 0,Y 336.042,Z 1079.518,A -85,B 0,C 180,E1 23253.995,E2 23253.995} C_VEL
LIN {X 0,Y 314.209,Z 1113.299,A -85,B 0,C 180,E1 23260.757,E2 23260.757} C_VEL
LIN {X 0,Y 296.304,Z 1140.341,A -85,B 0,C 180,E1 23268.47,E2 23268.47} C_VEL
LIN {X 0,Y 282.386,Z 1162.819,A -85,B 0,C 180,E1 23277.646,E2 23277.646} C_VEL
LIN {X 0,Y 274.398,Z 1178.893,A -85,B 0,C 180,E1 23287.324,E2 23287.324} C_VEL
LIN {X 0,Y 271.314,Z 1187.912,A -85,B 0,C 180,E1 23295.483,E2 23295.483} C_VEL
LIN {X 0,Y 270.441,Z 1193.135,A -85,B 0,C 180,E1 23303.582,E2 23303.582} C_VEL
LIN {X 0,Y 270.844,Z 1194.635,A -85,B 0,C 180,E1 23309.998,E2 23309.998} C_VEL
LIN {X 0,Y 270.393,Z 1193.707,A -85,B 0,C 180,E1 23316.416,E2 23316.416} C_VEL
LIN {X 0,Y 271.232,Z 1189.38,A -85,B 0,C 180,E1 23324.518,E2 23324.518} C_VEL
LIN {X 0,Y 275.352,Z 1179.509,A -85,B 0,C 180,E1 23334.23,E2 23334.23} C_VEL
LIN {X 0,Y 285.553,Z 1162.919,A -85,B 0,C 180,E1 23344.651,E2 23344.651} C_VEL
LIN {X 0,Y 301.833,Z 1140.809,A -85,B 0,C 180,E1 23353.864,E2 23353.864} C_VEL
LIN {X 0,Y 323.569,Z 1113.122,A -85,B 0,C 180,E1 23361.807,E2 23361.807} C_VEL
LIN {X 0,Y 349.251,Z 1078.933,A -85,B 0,C 180,E1 23368.463,E2 23368.463} C_VEL
LIN {X 0,Y 372.917,Z 1044.688,A -85,B 0,C 180,E1 23373.057,E2 23373.057} C_VEL
LIN {X 0,Y 397.316,Z 1004.12,A -85,B 0,C 180,E1 23376.914,E2 23376.914} C_VEL
LIN {X 0,Y 416.969,Z 965.26,A -85,B 0,C 180,E1 23379.591,E2 23379.591} C_VEL
LIN {X 0,Y 414.774,Z 950.859,A -85,B 0,C 180,E1 23384.148,E2 23384.148} C_VEL
LIN {X 0,Y 412.338,Z 939.445,A -85,B 0,C 180,E1 23389.447,E2 23389.447} C_VEL
LIN {X 0,Y 410.868,Z 932.101,A -85,B 0,C 180,E1 23395.787,E2 23395.787} C_VEL
LIN {X 0,Y 410.509,Z 931.726,A -85,B 0,C 180,E1 23400.006,E2 23400.006} C_VEL
LIN {X 0,Y 410.281,Z 938.609,A -85,B 0,C 180,E1 23406.092,E2 23406.092} C_VEL
LIN {X 0,Y 409.103,Z 943.833,A -85,B 0,C 180,E1 23407.771,E2 23407.771} C_VEL
LIN {X 0,Y 406.651,Z 954.207,A -85,B 0,C 180,E1 23410.495,E2 23410.495} C_VEL
LIN {X 0,Y 406.804,Z 968.663,A -85,B 0,C 180,E1 23415.758,E2 23415.758} C_VEL
LIN {X 0,Y 382.236,Z 1010.262,A -85,B 0,C 180,E1 23419.359,E2 23419.359} C_VEL
LIN {X 0,Y 357.53,Z 1044.882,A -85,B 0,C 180,E1 23423.667,E2 23423.667} C_VEL
LIN {X 0,Y 333.892,Z 1073.954,A -85,B 0,C 180,E1 23428.855,E2 23428.855} C_VEL
LIN {X 0,Y 309.757,Z 1100.4,A -85,B 0,C 180,E1 23435.843,E2 23435.843} C_VEL
LIN {X 0,Y 289.916,Z 1120.978,A -85,B 0,C 180,E1 23444.065,E2 23444.065} C_VEL
LIN {X 0,Y 274.998,Z 1136.462,A -85,B 0,C 180,E1 23453.794,E2 23453.794} C_VEL
LIN {X 0,Y 267.16,Z 1145.399,A -85,B 0,C 180,E1 23463.098,E2 23463.098} C_VEL
LIN {X 0,Y 263.211,Z 1150.167,A -85,B 0,C 180,E1 23473.32,E2 23473.32} C_VEL
LIN {X 0,Y 262.534,Z 1150.785,A -85,B 0,C 180,E1 23480.058,E2 23480.058} C_VEL
LIN {X 0,Y 263.18,Z 1149.337,A -85,B 0,C 180,E1 23486.71,E2 23486.71} C_VEL
LIN {X 0,Y 265.112,Z 1144.88,A -85,B 0,C 180,E1 23494.743,E2 23494.743} C_VEL
LIN {X 0,Y 269.472,Z 1137,A -85,B 0,C 180,E1 23502.964,E2 23502.964} C_VEL
LIN {X 0,Y 278.952,Z 1123.069,A -85,B 0,C 180,E1 23512.286,E2 23512.286} C_VEL
LIN {X 0,Y 293.994,Z 1103.491,A -85,B 0,C 180,E1 23520.932,E2 23520.932} C_VEL
LIN {X 0,Y 312.187,Z 1079.657,A -85,B 0,C 180,E1 23528.111,E2 23528.111} C_VEL
LIN {X 0,Y 334.152,Z 1049.041,A -85,B 0,C 180,E1 23534.505,E2 23534.505} C_VEL
LIN {X 0,Y 355.7,Z 1015.053,A -85,B 0,C 180,E1 23539.412,E2 23539.412} C_VEL
LIN {X 0,Y 376.326,Z 977.625,A -85,B 0,C 180,E1 23543.24,E2 23543.24} C_VEL
LIN {X 0,Y 387.163,Z 954.567,A -85,B 0,C 180,E1 23545.051,E2 23545.051} C_VEL
LIN {X 0,Y 385.007,Z 933.592,A -85,B 0,C 180,E1 23550.308,E2 23550.308} C_VEL
LIN {X 0,Y 381.591,Z 915.986,A -85,B 0,C 180,E1 23556.045,E2 23556.045} C_VEL
LIN {X 0,Y 378.726,Z 904.3,A -85,B 0,C 180,E1 23561.378,E2 23561.378} C_VEL
LIN {X 0,Y 376.792,Z 894.878,A -85,B 0,C 180,E1 23568.426,E2 23568.426} C_VEL
LIN {X 0,Y 377.011,Z 893.855,A -85,B 0,C 180,E1 23575.396,E2 23575.396} C_VEL
LIN {X 0,Y 378.262,Z 895.651,A -85,B 0,C 180,E1 23578.848,E2 23578.848} C_VEL
LIN {X 0,Y 381.101,Z 904.216,A -85,B 0,C 180,E1 23584.542,E2 23584.542} C_VEL
LIN {X 0,Y 385.337,Z 917.681,A -85,B 0,C 180,E1 23590.158,E2 23590.158} C_VEL
LIN {X 0,Y 390.176,Z 936.735,A -85,B 0,C 180,E1 23595.724,E2 23595.724} C_VEL
LIN {X 0,Y 394.092,Z 959.09,A -85,B 0,C 180,E1 23600.768,E2 23600.768} C_VEL
LIN {X 0,Y 374.615,Z 1002.778,A -85,B 0,C 180,E1 23603.857,E2 23603.857} C_VEL
LIN {X 0,Y 351.964,Z 1044.691,A -85,B 0,C 180,E1 23608.076,E2 23608.076} C_VEL
LIN {X 0,Y 330.259,Z 1079.926,A -85,B 0,C 180,E1 23613.064,E2 23613.064} C_VEL
LIN {X 0,Y 307.465,Z 1114.073,A -85,B 0,C 180,E1 23620.015,E2 23620.015} C_VEL
LIN {X 0,Y 288.575,Z 1141.455,A -85,B 0,C 180,E1 23628.112,E2 23628.112} C_VEL
LIN {X 0,Y 275.361,Z 1161.904,A -85,B 0,C 180,E1 23636.715,E2 23636.715} C_VEL
LIN {X 0,Y 267.592,Z 1176.566,A -85,B 0,C 180,E1 23645.455,E2 23645.455} C_VEL
LIN {X 0,Y 263.52,Z 1187.171,A -85,B 0,C 180,E1 23655.044,E2 23655.044} C_VEL
LIN {X 0,Y 262.551,Z 1192.45,A -85,B 0,C 180,E1 23663.388,E2 23663.388} C_VEL
LIN {X 0,Y 262.962,Z 1193.974,A -85,B 0,C 180,E1 23669.998,E2 23669.998} C_VEL
LIN {X 0,Y 262.493,Z 1193.079,A -85,B 0,C 180,E1 23676.61,E2 23676.61} C_VEL
LIN {X 0,Y 263.444,Z 1188.785,A -85,B 0,C 180,E1 23684.957,E2 23684.957} C_VEL
LIN {X 0,Y 267.602,Z 1179.449,A -85,B 0,C 180,E1 23694.551,E2 23694.551} C_VEL
LIN {X 0,Y 278.674,Z 1162.466,A -85,B 0,C 180,E1 23705.585,E2 23705.585} C_VEL
LIN {X 0,Y 295.864,Z 1140.292,A -85,B 0,C 180,E1 23715.016,E2 23715.016} C_VEL
LIN {X 0,Y 317.776,Z 1113.604,A -85,B 0,C 180,E1 23722.795,E2 23722.795} C_VEL
LIN {X 0,Y 343.309,Z 1080.841,A -85,B 0,C 180,E1 23729.275,E2 23729.275} C_VEL
LIN {X 0,Y 368.514,Z 1045.667,A -85,B 0,C 180,E1 23734.065,E2 23734.065} C_VEL
LIN {X 0,Y 394.004,Z 1004.396,A -85,B 0,C 180,E1 23737.964,E2 23737.964} C_VEL
LIN {X 0,Y 412.174,Z 969.475,A -85,B 0,C 180,E1 23740.407,E2 23740.407} C_VEL
LIN {X 0,Y 410.298,Z 955.6,A -85,B 0,C 180,E1 23745.065,E2 23745.065} C_VEL
LIN {X 0,Y 408.333,Z 945.1,A -85,B 0,C 180,E1 23750.419,E2 23750.419} C_VEL
LIN {X 0,Y 407.322,Z 939.261,A -85,B 0,C 180,E1 23755.751,E2 23755.751} C_VEL
LIN {X 0,Y 406.967,Z 938.861,A -85,B 0,C 180,E1 23760.006,E2 23760.006} C_VEL
LIN {X 0,Y 406.348,Z 946.185,A -85,B 0,C 180,E1 23766.412,E2 23766.412} C_VEL
LIN {X 0,Y 406.651,Z 954.207,A -85,B 0,C 180,E1 23770.495,E2 23770.495} C_VEL
LIN {X 0,Y 405.416,Z 960.222,A -85,B 0,C 180,E1 23772.129,E2 23772.129} C_VEL
LIN {X 0,Y 402.132,Z 972.315,A -85,B 0,C 180,E1 23774.732,E2 23774.732} C_VEL
LIN {X 0,Y 400.953,Z 975.28,A -85,B 0,C 180,E1 23775.189,E2 23775.189} C_VEL
LIN {X 0,Y 377.719,Z 1012.982,A -85,B 0,C 180,E1 23778.454,E2 23778.454} C_VEL
LIN {X 0,Y 350.879,Z 1049.252,A -85,B 0,C 180,E1 23783.064,E2 23783.064} C_VEL
LIN {X 0,Y 325.369,Z 1079.043,A -85,B 0,C 180,E1 23788.659,E2 23788.659} C_VEL
LIN {X 0,Y 300.958,Z 1104.768,A -85,B 0,C 180,E1 23795.889,E2 23795.889} C_VEL
LIN {X 0,Y 281.091,Z 1124.23,A -85,B 0,C 180,E1 23804.35,E2 23804.35} C_VEL
LIN {X 0,Y 267.236,Z 1138.002,A -85,B 0,C 180,E1 23813.579,E2 23813.579} C_VEL
LIN {X 0,Y 258.409,Z 1147.439,A -85,B 0,C 180,E1 23824.662,E2 23824.662} C_VEL
LIN {X 0,Y 255.433,Z 1150.783,A -85,B 0,C 180,E1 23832.796,E2 23832.796} C_VEL
LIN {X 0,Y 254.761,Z 1151.053,A -85,B 0,C 180,E1 23843.189,E2 23843.189} C_VEL
LIN {X 0,Y 256.005,Z 1148.57,A -85,B 0,C 180,E1 23850.002,E2 23850.002} C_VEL
LIN {X 0,Y 259.659,Z 1141.381,A -85,B 0,C 180,E1 23860.056,E2 23860.056} C_VEL
LIN {X 0,Y 267.654,Z 1129.213,A -85,B 0,C 180,E1 23869.802,E2 23869.802} C_VEL
LIN {X 0,Y 281.427,Z 1111.773,A -85,B 0,C 180,E1 23878.9,E2 23878.9} C_VEL
LIN {X 0,Y 300.464,Z 1087.921,A -85,B 0,C 180,E1 23887.124,E2 23887.124} C_VEL
LIN {X 0,Y 322.075,Z 1059.468,A -85,B 0,C 180,E1 23893.794,E2 23893.794} C_VEL
LIN {X 0,Y 345.928,Z 1024.467,A -85,B 0,C 180,E1 23899.378,E2 23899.378} C_VEL
LIN {X 0,Y 367.08,Z 988.134,A -85,B 0,C 180,E1 23903.414,E2 23903.414} C_VEL
LIN {X 0,Y 382.08,Z 957.493,A -85,B 0,C 180,E1 23906.03,E2 23906.03} C_VEL
LIN {X 0,Y 380.169,Z 936.795,A -85,B 0,C 180,E1 23911.503,E2 23911.503} C_VEL
LIN {X 0,Y 377.157,Z 919.47,A -85,B 0,C 180,E1 23917.619,E2 23917.619} C_VEL
LIN {X 0,Y 374.651,Z 908.127,A -85,B 0,C 180,E1 23923.593,E2 23923.593} C_VEL
LIN {X 0,Y 373.902,Z 902.402,A -85,B 0,C 180,E1 23928.335,E2 23928.335} C_VEL
LIN {X 0,Y 374.14,Z 901.205,A -85,B 0,C 180,E1 23935.36,E2 23935.36} C_VEL
LIN {X 0,Y 375.341,Z 903.109,A -85,B 0,C 180,E1 23938.839,E2 23938.839} C_VEL
LIN {X 0,Y 378.025,Z 911.811,A -85,B 0,C 180,E1 23944.579,E2 23944.579} C_VEL
LIN {X 0,Y 381.908,Z 925.519,A -85,B 0,C 180,E1 23950.25,E2 23950.25} C_VEL
LIN {X 0,Y 386.23,Z 944.94,A -85,B 0,C 180,E1 23955.889,E2 23955.889} C_VEL
LIN {X 0,Y 388.904,Z 962.702,A -85,B 0,C 180,E1 23959.966,E2 23959.966} C_VEL
LIN {X 0,Y 369.391,Z 1004.734,A -85,B 0,C 180,E1 23962.983,E2 23962.983} C_VEL
LIN {X 0,Y 345.796,Z 1047.104,A -85,B 0,C 180,E1 23967.305,E2 23967.305} C_VEL
LIN {X 0,Y 322.771,Z 1082.998,A -85,B 0,C 180,E1 23972.57,E2 23972.57} C_VEL
LIN {X 0,Y 300.358,Z 1115.403,A -85,B 0,C 180,E1 23979.386,E2 23979.386} C_VEL
LIN {X 0,Y 280.104,Z 1143.616,A -85,B 0,C 180,E1 23988.114,E2 23988.114} C_VEL
LIN {X 0,Y 266.528,Z 1164.029,A -85,B 0,C 180,E1 23997.343,E2 23997.343} C_VEL
LIN {X 0,Y 258.348,Z 1179.404,A -85,B 0,C 180,E1 24007.652,E2 24007.652} C_VEL
LIN {X 0,Y 255.198,Z 1188.66,A -85,B 0,C 180,E1 24017.469,E2 24017.469} C_VEL
LIN {X 0,Y 254.763,Z 1192.879,A -85,B 0,C 180,E1 24026.598,E2 24026.598} C_VEL
LIN {X 0,Y 254.842,Z 1193.152,A -85,B 0,C 180,E1 24033.398,E2 24033.398} C_VEL
LIN {X 0,Y 254.752,Z 1191.207,A -85,B 0,C 180,E1 24040.249,E2 24040.249} C_VEL
LIN {X 0,Y 257.176,Z 1184.538,A -85,B 0,C 180,E1 24049.949,E2 24049.949} C_VEL
LIN {X 0,Y 263.982,Z 1172.669,A -85,B 0,C 180,E1 24060.056,E2 24060.056} C_VEL
LIN {X 0,Y 278.465,Z 1153.763,A -85,B 0,C 180,E1 24070.63,E2 24070.63} C_VEL
LIN {X 0,Y 299.359,Z 1128.909,A -85,B 0,C 180,E1 24079.758,E2 24079.758} C_VEL
LIN {X 0,Y 323.114,Z 1100.828,A -85,B 0,C 180,E1 24086.774,E2 24086.774} C_VEL
LIN {X 0,Y 349.253,Z 1067.292,A -85,B 0,C 180,E1 24092.475,E2 24092.475} C_VEL
LIN {X 0,Y 374.749,Z 1030.913,A -85,B 0,C 180,E1 24096.763,E2 24096.763} C_VEL
LIN {X 0,Y 398.559,Z 991.045,A -85,B 0,C 180,E1 24100.007,E2 24100.007} C_VEL
LIN {X 0,Y 407.112,Z 974.791,A -85,B 0,C 180,E1 24101.053,E2 24101.053} C_VEL
LIN {X 0,Y 406.305,Z 963.062,A -85,B 0,C 180,E1 24104.915,E2 24104.915} C_VEL
LIN {X 0,Y 404.767,Z 953.922,A -85,B 0,C 180,E1 24109.247,E2 24109.247} C_VEL
LIN {X 0,Y 403.595,Z 946.298,A -85,B 0,C 180,E1 24115.711,E2 24115.711} C_VEL
LIN {X 0,Y 403.165,Z 945.857,A -85,B 0,C 180,E1 24120.006,E2 24120.006} C_VEL
LIN {X 0,Y 402.419,Z 953.325,A -85,B 0,C 180,E1 24126.474,E2 24126.474} C_VEL
LIN {X 0,Y 402.338,Z 964.554,A -85,B 0,C 180,E1 24131.929,E2 24131.929} C_VEL
LIN {X 0,Y 402.132,Z 972.315,A -85,B 0,C 180,E1 24134.732,E2 24134.732} C_VEL
LIN {X 0,Y 399.914,Z 976.805,A -85,B 0,C 180,E1 24135.192,E2 24135.192} C_VEL
LIN {X 0,Y 389.868,Z 990.367,A -85,B 0,C 180,E1 24135.231,E2 24135.231} C_VEL
LIN {X 0,Y 389.032,Z 991.653,A -85,B 0,C 180,E1 24135.314,E2 24135.314} C_VEL
LIN {X 0,Y 364.678,Z 1027.657,A -85,B 0,C 180,E1 24138.879,E2 24138.879} C_VEL
LIN {X 0,Y 337.602,Z 1061.319,A -85,B 0,C 180,E1 24143.765,E2 24143.765} C_VEL
LIN {X 0,Y 312.698,Z 1088.422,A -85,B 0,C 180,E1 24149.561,E2 24149.561} C_VEL
LIN {X 0,Y 288.794,Z 1111.992,A -85,B 0,C 180,E1 24157.176,E2 24157.176} C_VEL
LIN {X 0,Y 270.364,Z 1129.144,A -85,B 0,C 180,E1 24165.685,E2 24165.685} C_VEL
LIN {X 0,Y 256.256,Z 1142.62,A -85,B 0,C 180,E1 24176.532,E2 24176.532} C_VEL
LIN {X 0,Y 250.364,Z 1148.692,A -85,B 0,C 180,E1 24185.009,E2 24185.009} C_VEL
LIN {X 0,Y 247.071,Z 1152.004,A -85,B 0,C 180,E1 24195.841,E2 24195.841} C_VEL
LIN {X 0,Y 247.365,Z 1150.742,A -85,B 0,C 180,E1 24206.499,E2 24206.499} C_VEL
LIN {X 0,Y 249.515,Z 1146.303,A -85,B 0,C 180,E1 24215.214,E2 24215.214} C_VEL
LIN {X 0,Y 255.501,Z 1136.806,A -85,B 0,C 180,E1 24225.437,E2 24225.437} C_VEL
LIN {X 0,Y 268.049,Z 1120.639,A -85,B 0,C 180,E1 24235.949,E2 24235.949} C_VEL
LIN {X 0,Y 285.269,Z 1099.985,A -85,B 0,C 180,E1 24244.612,E2 24244.612} C_VEL
LIN {X 0,Y 307.228,Z 1072.982,A -85,B 0,C 180,E1 24252.194,E2 24252.194} C_VEL
LIN {X 0,Y 331.682,Z 1039.661,A -85,B 0,C 180,E1 24258.418,E2 24258.418} C_VEL
LIN {X 0,Y 354.017,Z 1004.715,A -85,B 0,C 180,E1 24262.911,E2 24262.911} C_VEL
LIN {X 0,Y 375.773,Z 964.623,A -85,B 0,C 180,E1 24266.519,E2 24266.519} C_VEL
LIN {X 0,Y 376.883,Z 962.25,A -85,B 0,C 180,E1 24266.688,E2 24266.688} C_VEL
LIN {X 0,Y 375.762,Z 943.135,A -85,B 0,C 180,E1 24271.794,E2 24271.794} C_VEL
LIN {X 0,Y 373.499,Z 927.267,A -85,B 0,C 180,E1 24277.416,E2 24277.416} C_VEL
LIN {X 0,Y 371.421,Z 915.683,A -85,B 0,C 180,E1 24283.446,E2 24283.446} C_VEL
LIN {X 0,Y 370.741,Z 909.843,A -85,B 0,C 180,E1 24288.234,E2 24288.234} C_VEL
LIN {X 0,Y 371.171,Z 908.525,A -85,B 0,C 180,E1 24295.323,E2 24295.323} C_VEL
LIN {X 0,Y 372.296,Z 910.502,A -85,B 0,C 180,E1 24298.831,E2 24298.831} C_VEL
LIN {X 0,Y 375.026,Z 920.468,A -85,B 0,C 180,E1 24305.195,E2 24305.195} C_VEL
LIN {X 0,Y 378.671,Z 935.019,A -85,B 0,C 180,E1 24310.921,E2 24310.921} C_VEL
LIN {X 0,Y 382.066,Z 953.176,A -85,B 0,C 180,E1 24316.067,E2 24316.067} C_VEL
LIN {X 0,Y 383.4,Z 967.347,A -85,B 0,C 180,E1 24319.215,E2 24319.215} C_VEL
LIN {X 0,Y 361.776,Z 1011.248,A -85,B 0,C 180,E1 24322.475,E2 24322.475} C_VEL
LIN {X 0,Y 339.109,Z 1050.247,A -85,B 0,C 180,E1 24326.601,E2 24326.601} C_VEL
LIN {X 0,Y 314.945,Z 1086.592,A -85,B 0,C 180,E1 24332.149,E2 24332.149} C_VEL
LIN {X 0,Y 293.12,Z 1116.809,A -85,B 0,C 180,E1 24338.783,E2 24338.783} C_VEL
LIN {X 0,Y 272.368,Z 1144.722,A -85,B 0,C 180,E1 24347.721,E2 24347.721} C_VEL
LIN {X 0,Y 258.48,Z 1164.709,A -85,B 0,C 180,E1 24357.262,E2 24357.262} C_VEL
LIN {X 0,Y 250.329,Z 1179.654,A -85,B 0,C 180,E1 24367.833,E2 24367.833} C_VEL
LIN {X 0,Y 247.244,Z 1188.508,A -85,B 0,C 180,E1 24377.892,E2 24377.892} C_VEL
LIN {X 0,Y 246.867,Z 1192.194,A -85,B 0,C 180,E1 24386.489,E2 24386.489} C_VEL
LIN {X 0,Y 247.202,Z 1192.651,A -85,B 0,C 180,E1 24389.998,E2 24389.998} C_VEL
LIN {X 0,Y 246.694,Z 1191.827,A -85,B 0,C 180,E1 24397.035,E2 24397.035} C_VEL
LIN {X 0,Y 247.855,Z 1187.593,A -85,B 0,C 180,E1 24405.922,E2 24405.922} C_VEL
LIN {X 0,Y 252.85,Z 1178.059,A -85,B 0,C 180,E1 24416.322,E2 24416.322} C_VEL
LIN {X 0,Y 265.086,Z 1161.671,A -85,B 0,C 180,E1 24427.535,E2 24427.535} C_VEL
LIN {X 0,Y 283.762,Z 1139.98,A -85,B 0,C 180,E1 24437.193,E2 24437.193} C_VEL
LIN {X 0,Y 307.932,Z 1112.824,A -85,B 0,C 180,E1 24445.281,E2 24445.281} C_VEL
LIN {X 0,Y 334.376,Z 1081.211,A -85,B 0,C 180,E1 24451.558,E2 24451.558} C_VEL
LIN {X 0,Y 361.733,Z 1045.214,A -85,B 0,C 180,E1 24456.407,E2 24456.407} C_VEL
LIN {X 0,Y 387.255,Z 1005.842,A -85,B 0,C 180,E1 24460.056,E2 24460.056} C_VEL
LIN {X 0,Y 402.672,Z 978.324,A -85,B 0,C 180,E1 24461.971,E2 24461.971} C_VEL
LIN {X 0,Y 401.417,Z 965.32,A -85,B 0,C 180,E1 24466.952,E2 24466.952} C_VEL
LIN {X 0,Y 399.992,Z 956.576,A -85,B 0,C 180,E1 24472.38,E2 24472.38} C_VEL
LIN {X 0,Y 399.742,Z 953.273,A -85,B 0,C 180,E1 24475.67,E2 24475.67} C_VEL
LIN {X 0,Y 399.633,Z 952.335,A -85,B 0,C 180,E1 24477.839,E2 24477.839} C_VEL
LIN {X 0,Y 398.953,Z 953.837,A -85,B 0,C 180,E1 24481.091,E2 24481.091} C_VEL
LIN {X 0,Y 398.198,Z 960.332,A -85,B 0,C 180,E1 24486.543,E2 24486.543} C_VEL
LIN {X 0,Y 397.767,Z 971.754,A -85,B 0,C 180,E1 24492.05,E2 24492.05} C_VEL
LIN {X 0,Y 397.09,Z 978.233,A -85,B 0,C 180,E1 24494.273,E2 24494.273} C_VEL
LIN {X 0,Y 389.032,Z 991.653,A -85,B 0,C 180,E1 24495.314,E2 24495.314} C_VEL
LIN {X 0,Y 379.009,Z 1005.463,A -85,B 0,C 180,E1 24495.929,E2 24495.929} C_VEL
LIN {X 0,Y 368.549,Z 1018.737,A -85,B 0,C 180,E1 24496.631,E2 24496.631} C_VEL
LIN {X 0,Y 341.848,Z 1052.873,A -85,B 0,C 180,E1 24501.009,E2 24501.009} C_VEL
LIN {X 0,Y 314.216,Z 1082.948,A -85,B 0,C 180,E1 24506.785,E2 24506.785} C_VEL
LIN {X 0,Y 290.142,Z 1106.46,A -85,B 0,C 180,E1 24513.562,E2 24513.562} C_VEL
LIN {X 0,Y 267.499,Z 1126.811,A -85,B 0,C 180,E1 24522.747,E2 24522.747} C_VEL
LIN {X 0,Y 251.682,Z 1140.804,A -85,B 0,C 180,E1 24533.103,E2 24533.103} C_VEL
LIN {X 0,Y 242.866,Z 1149.251,A -85,B 0,C 180,E1 24544.182,E2 24544.182} C_VEL
LIN {X 0,Y 239.248,Z 1152.651,A -85,B 0,C 180,E1 24555.368,E2 24555.368} C_VEL
LIN {X 0,Y 238.944,Z 1152.395,A -85,B 0,C 180,E1 24562.735,E2 24562.735} C_VEL
LIN {X 0,Y 240.224,Z 1150.04,A -85,B 0,C 180,E1 24570.002,E2 24570.002} C_VEL
LIN {X 0,Y 244.244,Z 1142.981,A -85,B 0,C 180,E1 24580.698,E2 24580.698} C_VEL
LIN {X 0,Y 252.953,Z 1131.052,A -85,B 0,C 180,E1 24591.006,E2 24591.006} C_VEL
LIN {X 0,Y 269.287,Z 1112.138,A -85,B 0,C 180,E1 24601.272,E2 24601.272} C_VEL
LIN {X 0,Y 291.128,Z 1086.801,A -85,B 0,C 180,E1 24609.968,E2 24609.968} C_VEL
LIN {X 0,Y 313.238,Z 1059.085,A -85,B 0,C 180,E1 24616.357,E2 24616.357} C_VEL
LIN {X 0,Y 337.273,Z 1025.571,A -85,B 0,C 180,E1 24621.637,E2 24621.637} C_VEL
LIN {X 0,Y 358.93,Z 990.131,A -85,B 0,C 180,E1 24625.53,E2 24625.53} C_VEL
LIN {X 0,Y 372.048,Z 964.925,A -85,B 0,C 180,E1 24627.752,E2 24627.752} C_VEL
LIN {X 0,Y 370.98,Z 945.401,A -85,B 0,C 180,E1 24633.372,E2 24633.372} C_VEL
LIN {X 0,Y 369.192,Z 930.849,A -85,B 0,C 180,E1 24639.035,E2 24639.035} C_VEL
LIN {X 0,Y 367.827,Z 921.507,A -85,B 0,C 180,E1 24644.505,E2 24644.505} C_VEL
LIN {X 0,Y 367.509,Z 917.253,A -85,B 0,C 180,E1 24648.129,E2 24648.129} C_VEL
LIN {X 0,Y 367.524,Z 915.603,A -85,B 0,C 180,E1 24653.275,E2 24653.275} C_VEL
LIN {X 0,Y 368.783,Z 916.565,A -85,B 0,C 180,E1 24657.645,E2 24657.645} C_VEL
LIN {X 0,Y 371.094,Z 925.626,A -85,B 0,C 180,E1 24664.08,E2 24664.08} C_VEL
LIN {X 0,Y 374.164,Z 939.331,A -85,B 0,C 180,E1 24669.877,E2 24669.877} C_VEL
LIN {X 0,Y 377.283,Z 957.959,A -85,B 0,C 180,E1 24675.412,E2 24675.412} C_VEL
LIN {X 0,Y 378.581,Z 969.734,A -85,B 0,C 180,E1 24678.254,E2 24678.254} C_VEL
LIN {X 0,Y 355.336,Z 1015.693,A -85,B 0,C 180,E1 24681.77,E2 24681.77} C_VEL
LIN {X 0,Y 332.004,Z 1053.991,A -85,B 0,C 180,E1 24685.98,E2 24685.98} C_VEL
LIN {X 0,Y 308.146,Z 1088.694,A -85,B 0,C 180,E1 24691.428,E2 24691.428} C_VEL
LIN {X 0,Y 284.99,Z 1119.408,A -85,B 0,C 180,E1 24698.477,E2 24698.477} C_VEL
LIN {X 0,Y 265.427,Z 1144.761,A -85,B 0,C 180,E1 24706.905,E2 24706.905} C_VEL
LIN {X 0,Y 250.511,Z 1165.286,A -85,B 0,C 180,E1 24717.117,E2 24717.117} C_VEL
LIN {X 0,Y 242.289,Z 1179.9,A -85,B 0,C 180,E1 24728.022,E2 24728.022} C_VEL
LIN {X 0,Y 239.4,Z 1187.782,A -85,B 0,C 180,E1 24737.489,E2 24737.489} C_VEL
LIN {X 0,Y 238.979,Z 1191.508,A -85,B 0,C 180,E1 24746.373,E2 24746.373} C_VEL
LIN {X 0,Y 239.336,Z 1191.991,A -85,B 0,C 180,E1 24749.998,E2 24749.998} C_VEL
LIN {X 0,Y 238.812,Z 1191.202,A -85,B 0,C 180,E1 24757.269,E2 24757.269} C_VEL
LIN {X 0,Y 240.102,Z 1187,A -85,B 0,C 180,E1 24766.45,E2 24766.45} C_VEL
LIN {X 0,Y 245.455,Z 1177.497,A -85,B 0,C 180,E1 24777.18,E2 24777.18} C_VEL
LIN {X 0,Y 258.677,Z 1160.997,A -85,B 0,C 180,E1 24788.751,E2 24788.751} C_VEL
LIN {X 0,Y 278.91,Z 1138.744,A -85,B 0,C 180,E1 24798.739,E2 24798.739} C_VEL
LIN {X 0,Y 304.806,Z 1110.807,A -85,B 0,C 180,E1 24806.96,E2 24806.96} C_VEL
LIN {X 0,Y 333.824,Z 1076.97,A -85,B 0,C 180,E1 24813.446,E2 24813.446} C_VEL
LIN {X 0,Y 361.169,Z 1041.228,A -85,B 0,C 180,E1 24818.014,E2 24818.014} C_VEL
LIN {X 0,Y 386.549,Z 1002.591,A -85,B 0,C 180,E1 24821.419,E2 24821.419} C_VEL
LIN {X 0,Y 397.629,Z 983.493,A -85,B 0,C 180,E1 24822.701,E2 24822.701} C_VEL
LIN {X 0,Y 397.255,Z 973.718,A -85,B 0,C 180,E1 24826.252,E2 24826.252} C_VEL
LIN {X 0,Y 396.215,Z 964.819,A -85,B 0,C 180,E1 24831.231,E2 24831.231} C_VEL
LIN {X 0,Y 395.83,Z 960.241,A -85,B 0,C 180,E1 24835.627,E2 24835.627} C_VEL
LIN {X 0,Y 395.76,Z 959.22,A -85,B 0,C 180,E1 24837.818,E2 24837.818} C_VEL
LIN {X 0,Y 395.315,Z 959.752,A -85,B 0,C 180,E1 24840.006,E2 24840.006} C_VEL
LIN {X 0,Y 394.099,Z 965.557,A -85,B 0,C 180,E1 24845.506,E2 24845.506} C_VEL
LIN {X 0,Y 393.265,Z 976.146,A -85,B 0,C 180,E1 24851.083,E2 24851.083} C_VEL
LIN {X 0,Y 392.789,Z 981.996,A -85,B 0,C 180,E1 24853.353,E2 24853.353} C_VEL
LIN {X 0,Y 368.549,Z 1018.737,A -85,B 0,C 180,E1 24856.631,E2 24856.631} C_VEL
LIN {X 0,Y 357.708,Z 1031.62,A -85,B 0,C 180,E1 24857.437,E2 24857.437} C_VEL
LIN {X 0,Y 347.87,Z 1042.46,A -85,B 0,C 180,E1 24858.195,E2 24858.195} C_VEL
LIN {X 0,Y 346.644,Z 1043.861,A -85,B 0,C 180,E1 24858.381,E2 24858.381} C_VEL
LIN {X 0,Y 318.598,Z 1075.043,A -85,B 0,C 180,E1 24863.609,E2 24863.609} C_VEL
LIN {X 0,Y 292.483,Z 1100.383,A -85,B 0,C 180,E1 24870.035,E2 24870.035} C_VEL
LIN {X 0,Y 268.774,Z 1121.338,A -85,B 0,C 180,E1 24878.216,E2 24878.216} C_VEL
LIN {X 0,Y 249.731,Z 1137.25,A -85,B 0,C 180,E1 24888.273,E2 24888.273} C_VEL
LIN {X 0,Y 237.863,Z 1147.626,A -85,B 0,C 180,E1 24899.456,E2 24899.456} C_VEL
LIN {X 0,Y 233.502,Z 1151.479,A -85,B 0,C 180,E1 24907.154,E2 24907.154} C_VEL
LIN {X 0,Y 231.077,Z 1153.467,A -85,B 0,C 180,E1 24918.852,E2 24918.852} C_VEL
LIN {X 0,Y 232.327,Z 1150.776,A -85,B 0,C 180,E1 24930.002,E2 24930.002} C_VEL
LIN {X 0,Y 235.513,Z 1145.236,A -85,B 0,C 180,E1 24939.232,E2 24939.232} C_VEL
LIN {X 0,Y 243.72,Z 1134.306,A -85,B 0,C 180,E1 24949.941,E2 24949.941} C_VEL
LIN {X 0,Y 258.091,Z 1118.03,A -85,B 0,C 180,E1 24959.848,E2 24959.848} C_VEL
LIN {X 0,Y 279.249,Z 1094.748,A -85,B 0,C 180,E1 24968.984,E2 24968.984} C_VEL
LIN {X 0,Y 304.504,Z 1064.782,A -85,B 0,C 180,E1 24976.536,E2 24976.536} C_VEL
LIN {X 0,Y 328.684,Z 1032.489,A -85,B 0,C 180,E1 24981.938,E2 24981.938} C_VEL
LIN {X 0,Y 351.771,Z 996.856,A -85,B 0,C 180,E1 24986.096,E2 24986.096} C_VEL
LIN {X 0,Y 366.442,Z 970.367,A -85,B 0,C 180,E1 24988.358,E2 24988.358} C_VEL
LIN {X 0,Y 366.902,Z 959.755,A -85,B 0,C 180,E1 24991.126,E2 24991.126} C_VEL
LIN {X 0,Y 365.937,Z 944.491,A -85,B 0,C 180,E1 24996.326,E2 24996.326} C_VEL
LIN {X 0,Y 364.722,Z 932.617,A -85,B 0,C 180,E1 25001.89,E2 25001.89} C_VEL
LIN {X 0,Y 364.138,Z 924.628,A -85,B 0,C 180,E1 25008.017,E2 25008.017} C_VEL
LIN {X 0,Y 364.501,Z 922.89,A -85,B 0,C 180,E1 25014.267,E2 25014.267} C_VEL
LIN {X 0,Y 365.798,Z 925.103,A -85,B 0,C 180,E1 25018.81,E2 25018.81} C_VEL
LIN {X 0,Y 367.766,Z 934.134,A -85,B 0,C 180,E1 25024.707,E2 25024.707} C_VEL
LIN {X 0,Y 370.357,Z 947.046,A -85,B 0,C 180,E1 25029.98,E2 25029.98} C_VEL
LIN {X 0,Y 372.738,Z 964.621,A -85,B 0,C 180,E1 25035.221,E2 25035.221} C_VEL
LIN {X 0,Y 373.292,Z 973.833,A -85,B 0,C 180,E1 25037.47,E2 25037.47} C_VEL
LIN {X 0,Y 350.527,Z 1017.183,A -85,B 0,C 180,E1 25040.776,E2 25040.776} C_VEL
LIN {X 0,Y 325.203,Z 1057.333,A -85,B 0,C 180,E1 25045.277,E2 25045.277} C_VEL
LIN {X 0,Y 301.292,Z 1090.748,A -85,B 0,C 180,E1 25050.698,E2 25050.698} C_VEL
LIN {X 0,Y 276.557,Z 1122.32,A -85,B 0,C 180,E1 25058.234,E2 25058.234} C_VEL
LIN {X 0,Y 256.413,Z 1147.262,A -85,B 0,C 180,E1 25067.144,E2 25067.144} C_VEL
LIN {X 0,Y 241.825,Z 1167.051,A -85,B 0,C 180,E1 25077.71,E2 25077.71} C_VEL
LIN {X 0,Y 234.703,Z 1179.089,A -85,B 0,C 180,E1 25087.273,E2 25087.273} C_VEL
LIN {X 0,Y 231.613,Z 1186.867,A -85,B 0,C 180,E1 25096.8,E2 25096.8} C_VEL
LIN {X 0,Y 231.082,Z 1190.821,A -85,B 0,C 180,E1 25106.249,E2 25106.249} C_VEL
LIN {X 0,Y 231.452,Z 1191.329,A -85,B 0,C 180,E1 25109.998,E2 25109.998} C_VEL
LIN {X 0,Y 230.915,Z 1190.577,A -85,B 0,C 180,E1 25117.519,E2 25117.519} C_VEL
LIN {X 0,Y 232.332,Z 1186.403,A -85,B 0,C 180,E1 25127.017,E2 25127.017} C_VEL
LIN {X 0,Y 238.462,Z 1176.489,A -85,B 0,C 180,E1 25138.482,E2 25138.482} C_VEL
LIN {X 0,Y 252.534,Z 1160.168,A -85,B 0,C 180,E1 25150.122,E2 25150.122} C_VEL
LIN {X 0,Y 273.482,Z 1138.306,A -85,B 0,C 180,E1 25160.053,E2 25160.053} C_VEL
LIN {X 0,Y 299.658,Z 1111.187,A -85,B 0,C 180,E1 25168.118,E2 25168.118} C_VEL
LIN {X 0,Y 328.225,Z 1079.033,A -85,B 0,C 180,E1 25174.359,E2 25174.359} C_VEL
LIN {X 0,Y 356.701,Z 1043.173,A -85,B 0,C 180,E1 25179.01,E2 25179.01} C_VEL
LIN {X 0,Y 383.509,Z 1003.409,A -85,B 0,C 180,E1 25182.499,E2 25182.499} C_VEL
LIN {X 0,Y 392.505,Z 988.348,A -85,B 0,C 180,E1 25183.505,E2 25183.505} C_VEL
LIN {X 0,Y 393.01,Z 983.903,A -85,B 0,C 180,E1 25184.862,E2 25184.862} C_VEL
LIN {X 0,Y 392.214,Z 973.349,A -85,B 0,C 180,E1 25190.022,E2 25190.022} C_VEL
LIN {X 0,Y 391.653,Z 967.06,A -85,B 0,C 180,E1 25195.58,E2 25195.58} C_VEL
LIN {X 0,Y 391.618,Z 965.97,A -85,B 0,C 180,E1 25197.795,E2 25197.795} C_VEL
LIN {X 0,Y 391.145,Z 966.541,A -85,B 0,C 180,E1 25200.006,E2 25200.006} C_VEL
LIN {X 0,Y 389.788,Z 972.488,A -85,B 0,C 180,E1 25205.568,E2 25205.568} C_VEL
LIN {X 0,Y 388.67,Z 981.909,A -85,B 0,C 180,E1 25210.649,E2 25210.649} C_VEL
LIN {X 0,Y 388.173,Z 986.095,A -85,B 0,C 180,E1 25212.371,E2 25212.371} C_VEL
LIN {X 0,Y 382.98,Z 994.579,A -85,B 0,C 180,E1 25213.194,E2 25213.194} C_VEL
LIN {X 0,Y 357.648,Z 1030.219,A -85,B 0,C 180,E1 25216.66,E2 25216.66} C_VEL
LIN {X 0,Y 346.644,Z 1043.861,A -85,B 0,C 180,E1 25218.381,E2 25218.381} C_VEL
LIN {X 0,Y 335.246,Z 1055.647,A -85,B 0,C 180,E1 25219.445,E2 25219.445} C_VEL
LIN {X 0,Y 323.561,Z 1066.84,A -85,B 0,C 180,E1 25220.603,E2 25220.603} C_VEL
LIN {X 0,Y 294.391,Z 1095.236,A -85,B 0,C 180,E1 25226.978,E2 25226.978} C_VEL
LIN {X 0,Y 269.547,Z 1116.866,A -85,B 0,C 180,E1 25234.535,E2 25234.535} C_VEL
LIN {X 0,Y 247.6,Z 1134.528,A -85,B 0,C 180,E1 25244.438,E2 25244.438} C_VEL
LIN {X 0,Y 232.327,Z 1146.727,A -85,B 0,C 180,E1 25256.438,E2 25256.438} C_VEL
LIN {X 0,Y 225.934,Z 1152.07,A -85,B 0,C 180,E1 25266.343,E2 25266.343} C_VEL
LIN {X 0,Y 223.207,Z 1154.151,A -85,B 0,C 180,E1 25278.284,E2 25278.284} C_VEL
LIN {X 0,Y 224.429,Z 1151.51,A -85,B 0,C 180,E1 25290.002,E2 25290.002} C_VEL
LIN {X 0,Y 227.763,Z 1146.036,A -85,B 0,C 180,E1 25299.549,E2 25299.549} C_VEL
LIN {X 0,Y 236.349,Z 1135.181,A -85,B 0,C 180,E1 25310.59,E2 25310.59} C_VEL
LIN {X 0,Y 251.31,Z 1119.028,A -85,B 0,C 180,E1 25320.739,E2 25320.739} C_VEL
LIN {X 0,Y 273.196,Z 1095.879,A -85,B 0,C 180,E1 25330.019,E2 25330.019} C_VEL
LIN {X 0,Y 298.036,Z 1067.405,A -85,B 0,C 180,E1 25337.326,E2 25337.326} C_VEL
LIN {X 0,Y 322.689,Z 1035.758,A -85,B 0,C 180,E1 25342.761,E2 25342.761} C_VEL
LIN {X 0,Y 347.133,Z 999.07,A -85,B 0,C 180,E1 25347.098,E2 25347.098} C_VEL
LIN {X 0,Y 361.666,Z 973.688,A -85,B 0,C 180,E1 25349.277,E2 25349.277} C_VEL
LIN {X 0,Y 362.084,Z 959.841,A -85,B 0,C 180,E1 25353.335,E2 25353.335} C_VEL
LIN {X 0,Y 361.381,Z 945.846,A -85,B 0,C 180,E1 25358.752,E2 25358.752} C_VEL
LIN {X 0,Y 360.637,Z 935.852,A -85,B 0,C 180,E1 25364.528,E2 25364.528} C_VEL
LIN {X 0,Y 360.56,Z 931.927,A -85,B 0,C 180,E1 25367.897,E2 25367.897} C_VEL
LIN {X 0,Y 360.865,Z 929.917,A -85,B 0,C 180,E1 25373.295,E2 25373.295} C_VEL
LIN {X 0,Y 362.061,Z 930.948,A -85,B 0,C 180,E1 25377.601,E2 25377.601} C_VEL
LIN {X 0,Y 363.864,Z 940.309,A -85,B 0,C 180,E1 25384.161,E2 25384.161} C_VEL
LIN {X 0,Y 365.989,Z 952.885,A -85,B 0,C 180,E1 25389.5,E2 25389.5} C_VEL
LIN {X 0,Y 367.947,Z 970.504,A -85,B 0,C 180,E1 25394.867,E2 25394.867} C_VEL
LIN {X 0,Y 367.921,Z 977.992,A -85,B 0,C 180,E1 25396.625,E2 25396.625} C_VEL
LIN {X 0,Y 345.371,Z 1019.272,A -85,B 0,C 180,E1 25399.826,E2 25399.826} C_VEL
LIN {X 0,Y 318.938,Z 1059.945,A -85,B 0,C 180,E1 25404.443,E2 25404.443} C_VEL
LIN {X 0,Y 293.595,Z 1093.839,A -85,B 0,C 180,E1 25410.156,E2 25410.156} C_VEL
LIN {X 0,Y 269.3,Z 1123.781,A -85,B 0,C 180,E1 25417.568,E2 25417.568} C_VEL
LIN {X 0,Y 248.391,Z 1148.599,A -85,B 0,C 180,E1 25426.877,E2 25426.877} C_VEL
LIN {X 0,Y 233.629,Z 1167.867,A -85,B 0,C 180,E1 25437.794,E2 25437.794} C_VEL
LIN {X 0,Y 225.666,Z 1181.114,A -85,B 0,C 180,E1 25449.606,E2 25449.606} C_VEL
LIN {X 0,Y 223.541,Z 1187.187,A -85,B 0,C 180,E1 25458.297,E2 25458.297} C_VEL
LIN {X 0,Y 223.183,Z 1190.135,A -85,B 0,C 180,E1 25466.116,E2 25466.116} C_VEL
LIN {X 0,Y 223.566,Z 1190.667,A -85,B 0,C 180,E1 25469.998,E2 25469.998} C_VEL
LIN {X 0,Y 223.044,Z 1189.954,A -85,B 0,C 180,E1 25477.786,E2 25477.786} C_VEL
LIN {X 0,Y 224.583,Z 1185.799,A -85,B 0,C 180,E1 25487.623,E2 25487.623} C_VEL
LIN {X 0,Y 231.151,Z 1176.043,A -85,B 0,C 180,E1 25499.358,E2 25499.358} C_VEL
LIN {X 0,Y 246.075,Z 1159.769,A -85,B 0,C 180,E1 25511.309,E2 25511.309} C_VEL
LIN {X 0,Y 268.196,Z 1137.876,A -85,B 0,C 180,E1 25521.421,E2 25521.421} C_VEL
LIN {X 0,Y 295.783,Z 1110.385,A -85,B 0,C 180,E1 25529.598,E2 25529.598} C_VEL
LIN {X 0,Y 325.73,Z 1077.635,A -85,B 0,C 180,E1 25535.847,E2 25535.847} C_VEL
LIN {X 0,Y 354.905,Z 1041.57,A -85,B 0,C 180,E1 25540.395,E2 25540.395} C_VEL
LIN {X 0,Y 381.665,Z 1002.586,A -85,B 0,C 180,E1 25543.708,E2 25543.708} C_VEL
LIN {X 0,Y 388.315,Z 991.496,A -85,B 0,C 180,E1 25544.516,E2 25544.516} C_VEL
LIN {X 0,Y 387.924,Z 980.671,A -85,B 0,C 180,E1 25549.665,E2 25549.665} C_VEL
LIN {X 0,Y 387.487,Z 973.861,A -85,B 0,C 180,E1 25555.533,E2 25555.533} C_VEL
LIN {X 0,Y 387.477,Z 972.715,A -85,B 0,C 180,E1 25557.771,E2 25557.771} C_VEL
LIN {X 0,Y 386.978,Z 973.326,A -85,B 0,C 180,E1 25560.006,E2 25560.006} C_VEL
LIN {X 0,Y 385.227,Z 979.247,A -85,B 0,C 180,E1 25565.634,E2 25565.634} C_VEL
LIN {X 0,Y 383.776,Z 988.874,A -85,B 0,C 180,E1 25570.786,E2 25570.786} C_VEL
LIN {X 0,Y 383.396,Z 990.961,A -85,B 0,C 180,E1 25571.66,E2 25571.66} C_VEL
LIN {X 0,Y 356.298,Z 1029.109,A -85,B 0,C 180,E1 25575.237,E2 25575.237} C_VEL
LIN {X 0,Y 327.239,Z 1062.852,A -85,B 0,C 180,E1 25579.92,E2 25579.92} C_VEL
LIN {X 0,Y 323.561,Z 1066.84,A -85,B 0,C 180,E1 25580.603,E2 25580.603} C_VEL
LIN {X 0,Y 311.612,Z 1077.52,A -85,B 0,C 180,E1 25581.932,E2 25581.932} C_VEL
LIN {X 0,Y 299.617,Z 1087.458,A -85,B 0,C 180,E1 25583.402,E2 25583.402} C_VEL
LIN {X 0,Y 273.377,Z 1110.243,A -85,B 0,C 180,E1 25590.211,E2 25590.211} C_VEL
LIN {X 0,Y 248.563,Z 1129.876,A -85,B 0,C 180,E1 25599.54,E2 25599.54} C_VEL
LIN {X 0,Y 229.701,Z 1143.975,A -85,B 0,C 180,E1 25611.152,E2 25611.152} C_VEL
LIN {X 0,Y 220.687,Z 1150.938,A -85,B 0,C 180,E1 25621.361,E2 25621.361} C_VEL
LIN {X 0,Y 215.809,Z 1154.6,A -85,B 0,C 180,E1 25633.737,E2 25633.737} C_VEL
LIN {X 0,Y 215.238,Z 1154.41,A -85,B 0,C 180,E1 25641.93,E2 25641.93} C_VEL
LIN {X 0,Y 216.529,Z 1152.244,A -85,B 0,C 180,E1 25650.002,E2 25650.002} C_VEL
LIN {X 0,Y 220.016,Z 1146.838,A -85,B 0,C 180,E1 25659.889,E2 25659.889} C_VEL
LIN {X 0,Y 229.007,Z 1136.057,A -85,B 0,C 180,E1 25671.282,E2 25671.282} C_VEL
LIN {X 0,Y 244.593,Z 1120.026,A -85,B 0,C 180,E1 25681.68,E2 25681.68} C_VEL
LIN {X 0,Y 267.247,Z 1096.97,A -85,B 0,C 180,E1 25691.098,E2 25691.098} C_VEL
LIN {X 0,Y 292.806,Z 1068.647,A -85,B 0,C 180,E1 25698.448,E2 25698.448} C_VEL
LIN {X 0,Y 316.878,Z 1038.868,A -85,B 0,C 180,E1 25703.637,E2 25703.637} C_VEL
LIN {X 0,Y 342.58,Z 1001.327,A -85,B 0,C 180,E1 25708.116,E2 25708.116} C_VEL
LIN {X 0,Y 357.02,Z 976.463,A -85,B 0,C 180,E1 25710.375,E2 25710.375} C_VEL
LIN {X 0,Y 357.415,Z 961.203,A -85,B 0,C 180,E1 25715.363,E2 25715.363} C_VEL
LIN {X 0,Y 357.113,Z 949.169,A -85,B 0,C 180,E1 25720.6,E2 25720.6} C_VEL
LIN {X 0,Y 356.865,Z 940.147,A -85,B 0,C 180,E1 25726.892,E2 25726.892} C_VEL
LIN {X 0,Y 357.082,Z 937.576,A -85,B 0,C 180,E1 25730.247,E2 25730.247} C_VEL
LIN {X 0,Y 357.783,Z 937.097,A -85,B 0,C 180,E1 25735.148,E2 25735.148} C_VEL
LIN {X 0,Y 358.668,Z 939.396,A -85,B 0,C 180,E1 25738.786,E2 25738.786} C_VEL
LIN {X 0,Y 360.251,Z 948.782,A -85,B 0,C 180,E1 25744.806,E2 25744.806} C_VEL
LIN {X 0,Y 362.058,Z 962.16,A -85,B 0,C 180,E1 25750.211,E2 25750.211} C_VEL
LIN {X 0,Y 363.302,Z 980.585,A -85,B 0,C 180,E1 25755.624,E2 25755.624} C_VEL
LIN {X 0,Y 340.158,Z 1021.609,A -85,B 0,C 180,E1 25758.871,E2 25758.871} C_VEL
LIN {X 0,Y 314.013,Z 1060.701,A -85,B 0,C 180,E1 25763.333,E2 25763.333} C_VEL
LIN {X 0,Y 286.761,Z 1095.929,A -85,B 0,C 180,E1 25769.384,E2 25769.384} C_VEL
LIN {X 0,Y 262.101,Z 1125.051,A -85,B 0,C 180,E1 25776.861,E2 25776.861} C_VEL
LIN {X 0,Y 240.813,Z 1149.406,A -85,B 0,C 180,E1 25786.347,E2 25786.347} C_VEL
LIN {X 0,Y 226.614,Z 1167.007,A -85,B 0,C 180,E1 25796.67,E2 25796.67} C_VEL
LIN {X 0,Y 218.594,Z 1179.304,A -85,B 0,C 180,E1 25807.651,E2 25807.651} C_VEL
LIN {X 0,Y 215.519,Z 1186.971,A -85,B 0,C 180,E1 25818.947,E2 25818.947} C_VEL
LIN {X 0,Y 215.284,Z 1189.446,A -85,B 0,C 180,E1 25825.973,E2 25825.973} C_VEL
LIN {X 0,Y 215.68,Z 1190.004,A -85,B 0,C 180,E1 25829.998,E2 25829.998} C_VEL
LIN {X 0,Y 215.148,Z 1189.33,A -85,B 0,C 180,E1 25838.073,E2 25838.073} C_VEL
LIN {X 0,Y 216.874,Z 1185.188,A -85,B 0,C 180,E1 25848.271,E2 25848.271} C_VEL
LIN {X 0,Y 223.956,Z 1175.484,A -85,B 0,C 180,E1 25860.399,E2 25860.399} C_VEL
LIN {X 0,Y 239.841,Z 1159.256,A -85,B 0,C 180,E1 25872.631,E2 25872.631} C_VEL
LIN {X 0,Y 261.969,Z 1138.477,A -85,B 0,C 180,E1 25882.469,E2 25882.469} C_VEL
LIN {X 0,Y 290.647,Z 1110.97,A -85,B 0,C 180,E1 25890.78,E2 25890.78} C_VEL
LIN {X 0,Y 320.473,Z 1079.574,A -85,B 0,C 180,E1 25896.847,E2 25896.847} C_VEL
LIN {X 0,Y 350.684,Z 1043.537,A -85,B 0,C 180,E1 25901.437,E2 25901.437} C_VEL
LIN {X 0,Y 377.503,Z 1005.588,A -85,B 0,C 180,E1 25904.669,E2 25904.669} C_VEL
LIN {X 0,Y 383.553,Z 996.101,A -85,B 0,C 180,E1 25905.361,E2 25905.361} C_VEL
LIN {X 0,Y 383.33,Z 986.381,A -85,B 0,C 180,E1 25910.234,E2 25910.234} C_VEL
LIN {X 0,Y 383.101,Z 980.536,A -85,B 0,C 180,E1 25915.481,E2 25915.481} C_VEL
LIN {X 0,Y 383.12,Z 979.345,A -85,B 0,C 180,E1 25917.746,E2 25917.746} C_VEL
LIN {X 0,Y 382.533,Z 979.929,A -85,B 0,C 180,E1 25920.006,E2 25920.006} C_VEL
LIN {X 0,Y 380.656,Z 986.023,A -85,B 0,C 180,E1 25925.703,E2 25925.703} C_VEL
LIN {X 0,Y 378.776,Z 995.398,A -85,B 0,C 180,E1 25930.757,E2 25930.757} C_VEL
LIN {X 0,Y 352.586,Z 1031.092,A -85,B 0,C 180,E1 25934.156,E2 25934.156} C_VEL
LIN {X 0,Y 323.155,Z 1064.398,A -85,B 0,C 180,E1 25938.755,E2 25938.755} C_VEL
LIN {X 0,Y 299.617,Z 1087.458,A -85,B 0,C 180,E1 25943.402,E2 25943.402} C_VEL
LIN {X 0,Y 287.432,Z 1096.894,A -85,B 0,C 180,E1 25945.048,E2 25945.048} C_VEL
LIN {X 0,Y 275.34,Z 1105.621,A -85,B 0,C 180,E1 25946.917,E2 25946.917} C_VEL
LIN {X 0,Y 250.929,Z 1124.672,A -85,B 0,C 180,E1 25954.783,E2 25954.783} C_VEL
LIN {X 0,Y 228.705,Z 1140.565,A -85,B 0,C 180,E1 25965.753,E2 25965.753} C_VEL
LIN {X 0,Y 215.596,Z 1149.976,A -85,B 0,C 180,E1 25977.278,E2 25977.278} C_VEL
LIN {X 0,Y 209.16,Z 1154.499,A -85,B 0,C 180,E1 25988.826,E2 25988.826} C_VEL
LIN {X 0,Y 207.475,Z 1155.442,A -85,B 0,C 180,E1 25997.381,E2 25997.381} C_VEL
LIN {X 0,Y 208.64,Z 1152.978,A -85,B 0,C 180,E1 26010.002,E2 26010.002} C_VEL
LIN {X 0,Y 212.291,Z 1147.637,A -85,B 0,C 180,E1 26020.253,E2 26020.253} C_VEL
LIN {X 0,Y 221.714,Z 1136.927,A -85,B 0,C 180,E1 26032.018,E2 26032.018} C_VEL
LIN {X 0,Y 237.948,Z 1121.023,A -85,B 0,C 180,E1 26042.673,E2 26042.673} C_VEL
LIN {X 0,Y 261.397,Z 1098.051,A -85,B 0,C 180,E1 26052.227,E2 26052.227} C_VEL
LIN {X 0,Y 286.511,Z 1071.264,A -85,B 0,C 180,E1 26059.306,E2 26059.306} C_VEL
LIN {X 0,Y 312.492,Z 1040.074,A -85,B 0,C 180,E1 26064.813,E2 26064.813} C_VEL
LIN {X 0,Y 338.574,Z 1002.922,A -85,B 0,C 180,E1 26069.226,E2 26069.226} C_VEL
LIN {X 0,Y 351.994,Z 981.086,A -85,B 0,C 180,E1 26071.126,E2 26071.126} C_VEL
LIN {X 0,Y 352.906,Z 966.509,A -85,B 0,C 180,E1 26076.021,E2 26076.021} C_VEL
LIN {X 0,Y 353.037,Z 953.837,A -85,B 0,C 180,E1 26081.913,E2 26081.913} C_VEL
LIN {X 0,Y 353.078,Z 946.356,A -85,B 0,C 180,E1 26087.636,E2 26087.636} C_VEL
LIN {X 0,Y 353.699,Z 944.028,A -85,B 0,C 180,E1 26093.322,E2 26093.322} C_VEL
LIN {X 0,Y 354.829,Z 945.106,A -85,B 0,C 180,E1 26097.552,E2 26097.552} C_VEL
LIN {X 0,Y 355.933,Z 953.586,A -85,B 0,C 180,E1 26103.645,E2 26103.645} C_VEL
LIN {X 0,Y 357.393,Z 966.166,A -85,B 0,C 180,E1 26109.117,E2 26109.117} C_VEL
LIN {X 0,Y 358.259,Z 984.054,A -85,B 0,C 180,E1 26114.653,E2 26114.653} C_VEL
LIN {X 0,Y 332.584,Z 1027.847,A -85,B 0,C 180,E1 26118.265,E2 26118.265} C_VEL
LIN {X 0,Y 306.627,Z 1064.765,A -85,B 0,C 180,E1 26122.694,E2 26122.694} C_VEL
LIN {X 0,Y 279.795,Z 1098.285,A -85,B 0,C 180,E1 26128.638,E2 26128.638} C_VEL
LIN {X 0,Y 254.609,Z 1126.701,A -85,B 0,C 180,E1 26136.247,E2 26136.247} C_VEL
LIN {X 0,Y 232.842,Z 1150.689,A -85,B 0,C 180,E1 26146.012,E2 26146.012} C_VEL
LIN {X 0,Y 217.679,Z 1168.625,A -85,B 0,C 180,E1 26157.45,E2 26157.45} C_VEL
LIN {X 0,Y 209.939,Z 1180.578,A -85,B 0,C 180,E1 26169.318,E2 26169.318} C_VEL
LIN {X 0,Y 207.857,Z 1185.748,A -85,B 0,C 180,E1 26177.4,E2 26177.4} C_VEL
LIN {X 0,Y 207.385,Z 1188.758,A -85,B 0,C 180,E1 26185.819,E2 26185.819} C_VEL
LIN {X 0,Y 207.815,Z 1189.344,A -85,B 0,C 180,E1 26189.998,E2 26189.998} C_VEL
LIN {X 0,Y 207.261,Z 1188.705,A -85,B 0,C 180,E1 26198.383,E2 26198.383} C_VEL
LIN {X 0,Y 209.807,Z 1183.581,A -85,B 0,C 180,E1 26210.587,E2 26210.587} C_VEL
LIN {X 0,Y 218.803,Z 1172.806,A -85,B 0,C 180,E1 26223.537,E2 26223.537} C_VEL
LIN {X 0,Y 235.898,Z 1156.822,A -85,B 0,C 180,E1 26235.212,E2 26235.212} C_VEL
LIN {X 0,Y 262.509,Z 1132.935,A -85,B 0,C 180,E1 26245.839,E2 26245.839} C_VEL
LIN {X 0,Y 290.925,Z 1106.474,A -85,B 0,C 180,E1 26253.187,E2 26253.187} C_VEL
LIN {X 0,Y 323.303,Z 1072.804,A -85,B 0,C 180,E1 26259.193,E2 26259.193} C_VEL
LIN {X 0,Y 352.512,Z 1037.639,A -85,B 0,C 180,E1 26263.275,E2 26263.275} C_VEL
LIN {X 0,Y 378.107,Z 1001.498,A -85,B 0,C 180,E1 26266.132,E2 26266.132} C_VEL
LIN {X 0,Y 378.816,Z 995.918,A -85,B 0,C 180,E1 26268.501,E2 26268.501} C_VEL
LIN {X 0,Y 378.542,Z 988.464,A -85,B 0,C 180,E1 26273.999,E2 26273.999} C_VEL
LIN {X 0,Y 378.679,Z 985.899,A -85,B 0,C 180,E1 26277.719,E2 26277.719} C_VEL
LIN {X 0,Y 377.791,Z 986.992,A -85,B 0,C 180,E1 26280.538,E2 26280.538} C_VEL
LIN {X 0,Y 375.851,Z 992.622,A -85,B 0,C 180,E1 26285.776,E2 26285.776} C_VEL
LIN {X 0,Y 374.182,Z 999.976,A -85,B 0,C 180,E1 26289.862,E2 26289.862} C_VEL
LIN {X 0,Y 345.522,Z 1037.211,A -85,B 0,C 180,E1 26293.538,E2 26293.538} C_VEL
LIN {X 0,Y 316.365,Z 1068.832,A -85,B 0,C 180,E1 26298.065,E2 26298.065} C_VEL
LIN {X 0,Y 285.483,Z 1097.197,A -85,B 0,C 180,E1 26304.355,E2 26304.355} C_VEL
LIN {X 0,Y 275.34,Z 1105.621,A -85,B 0,C 180,E1 26306.917,E2 26306.917} C_VEL
LIN {X 0,Y 263.296,Z 1113.78,A -85,B 0,C 180,E1 26309.004,E2 26309.004} C_VEL
LIN {X 0,Y 251.373,Z 1121.255,A -85,B 0,C 180,E1 26311.333,E2 26311.333} C_VEL
LIN {X 0,Y 227.023,Z 1138.241,A -85,B 0,C 180,E1 26321.746,E2 26321.746} C_VEL
LIN {X 0,Y 209.697,Z 1149.763,A -85,B 0,C 180,E1 26334.798,E2 26334.798} C_VEL
LIN {X 0,Y 201.535,Z 1155.124,A -85,B 0,C 180,E1 26347.984,E2 26347.984} C_VEL
LIN {X 0,Y 199.39,Z 1155.862,A -85,B 0,C 180,E1 26360.222,E2 26360.222} C_VEL
LIN {X 0,Y 200.735,Z 1153.711,A -85,B 0,C 180,E1 26370.002,E2 26370.002} C_VEL
LIN {X 0,Y 204.569,Z 1148.435,A -85,B 0,C 180,E1 26380.644,E2 26380.644} C_VEL
LIN {X 0,Y 214.461,Z 1137.798,A -85,B 0,C 180,E1 26392.804,E2 26392.804} C_VEL
LIN {X 0,Y 231.381,Z 1122.015,A -85,B 0,C 180,E1 26403.722,E2 26403.722} C_VEL
LIN {X 0,Y 256.761,Z 1098.105,A -85,B 0,C 180,E1 26413.753,E2 26413.753} C_VEL
LIN {X 0,Y 283.942,Z 1069.746,A -85,B 0,C 180,E1 26421.111,E2 26421.111} C_VEL
LIN {X 0,Y 310.532,Z 1038.249,A -85,B 0,C 180,E1 26426.447,E2 26426.447} C_VEL
LIN {X 0,Y 336.885,Z 1001.231,A -85,B 0,C 180,E1 26430.681,E2 26430.681} C_VEL
LIN {X 0,Y 347.311,Z 984.251,A -85,B 0,C 180,E1 26432.235,E2 26432.235} C_VEL
LIN {X 0,Y 348.362,Z 970.961,A -85,B 0,C 180,E1 26437.012,E2 26437.012} C_VEL
LIN {X 0,Y 348.792,Z 959.942,A -85,B 0,C 180,E1 26442.395,E2 26442.395} C_VEL
LIN {X 0,Y 349.184,Z 953.479,A -85,B 0,C 180,E1 26447.496,E2 26447.496} C_VEL
LIN {X 0,Y 349.768,Z 950.936,A -85,B 0,C 180,E1 26452.546,E2 26452.546} C_VEL
LIN {X 0,Y 350.956,Z 952.039,A -85,B 0,C 180,E1 26457.525,E2 26457.525} C_VEL
LIN {X 0,Y 351.949,Z 960.731,A -85,B 0,C 180,E1 26463.686,E2 26463.686} C_VEL
LIN {X 0,Y 352.89,Z 973.524,A -85,B 0,C 180,E1 26469.234,E2 26469.234} C_VEL
LIN {X 0,Y 352.998,Z 988.308,A -85,B 0,C 180,E1 26473.822,E2 26473.822} C_VEL
LIN {X 0,Y 328.15,Z 1029.197,A -85,B 0,C 180,E1 26477.154,E2 26477.154} C_VEL
LIN {X 0,Y 300.725,Z 1066.923,A -85,B 0,C 180,E1 26481.733,E2 26481.733} C_VEL
LIN {X 0,Y 273.212,Z 1100.081,A -85,B 0,C 180,E1 26487.751,E2 26487.751} C_VEL
LIN {X 0,Y 245.644,Z 1129.97,A -85,B 0,C 180,E1 26496.148,E2 26496.148} C_VEL
LIN {X 0,Y 225.131,Z 1151.522,A -85,B 0,C 180,E1 26505.503,E2 26505.503} C_VEL
LIN {X 0,Y 208.784,Z 1170.299,A -85,B 0,C 180,E1 26518.347,E2 26518.347} C_VEL
LIN {X 0,Y 201.484,Z 1181.406,A -85,B 0,C 180,E1 26530.657,E2 26530.657} C_VEL
LIN {X 0,Y 199.49,Z 1186.909,A -85,B 0,C 180,E1 26541.284,E2 26541.284} C_VEL
LIN {X 0,Y 199.925,Z 1188.681,A -85,B 0,C 180,E1 26549.998,E2 26549.998} C_VEL
LIN {X 0,Y 199.394,Z 1187.73,A -85,B 0,C 180,E1 26559.925,E2 26559.925} C_VEL
LIN {X 0,Y 202.394,Z 1182.661,A -85,B 0,C 180,E1 26571.918,E2 26571.918} C_VEL
LIN {X 0,Y 212.941,Z 1171.322,A -85,B 0,C 180,E1 26585.676,E2 26585.676} C_VEL
LIN {X 0,Y 231.286,Z 1155.23,A -85,B 0,C 180,E1 26597.307,E2 26597.307} C_VEL
LIN {X 0,Y 258.851,Z 1131.757,A -85,B 0,C 180,E1 26607.629,E2 26607.629} C_VEL
LIN {X 0,Y 288.234,Z 1105.184,A -85,B 0,C 180,E1 26614.882,E2 26614.882} C_VEL
LIN {X 0,Y 320.46,Z 1072.559,A -85,B 0,C 180,E1 26620.575,E2 26620.575} C_VEL
LIN {X 0,Y 351.055,Z 1036.459,A -85,B 0,C 180,E1 26624.653,E2 26624.653} C_VEL
LIN {X 0,Y 373.744,Z 1005.214,A -85,B 0,C 180,E1 26627.082,E2 26627.082} C_VEL
LIN {X 0,Y 373.943,Z 997.268,A -85,B 0,C 180,E1 26631.875,E2 26631.875} C_VEL
LIN {X 0,Y 374.172,Z 992.41,A -85,B 0,C 180,E1 26637.692,E2 26637.692} C_VEL
LIN {X 0,Y 373.44,Z 993.033,A -85,B 0,C 180,E1 26640.006,E2 26640.006} C_VEL
LIN {X 0,Y 370.972,Z 999.198,A -85,B 0,C 180,E1 26645.852,E2 26645.852} C_VEL
LIN {X 0,Y 369.547,Z 1004.392,A -85,B 0,C 180,E1 26648.897,E2 26648.897} C_VEL
LIN {X 0,Y 364.045,Z 1012.056,A -85,B 0,C 180,E1 26649.698,E2 26649.698} C_VEL
LIN {X 0,Y 336.888,Z 1045.049,A -85,B 0,C 180,E1 26653.091,E2 26653.091} C_VEL
LIN {X 0,Y 305.114,Z 1077.271,A -85,B 0,C 180,E1 26658.114,E2 26658.114} C_VEL
LIN {X 0,Y 276.321,Z 1102.2,A -85,B 0,C 180,E1 26664.149,E2 26664.149} C_VEL
LIN {X 0,Y 251.373,Z 1121.255,A -85,B 0,C 180,E1 26671.333,E2 26671.333} C_VEL
LIN {X 0,Y 239.656,Z 1128.129,A -85,B 0,C 180,E1 26673.923,E2 26673.923} C_VEL
LIN {X 0,Y 228.244,Z 1134.299,A -85,B 0,C 180,E1 26676.811,E2 26676.811} C_VEL
LIN {X 0,Y 207.595,Z 1147.411,A -85,B 0,C 180,E1 26689.073,E2 26689.073} C_VEL
LIN {X 0,Y 196.122,Z 1154.449,A -85,B 0,C 180,E1 26702.467,E2 26702.467} C_VEL
LIN {X 0,Y 192.55,Z 1156.553,A -85,B 0,C 180,E1 26711.707,E2 26711.707} C_VEL
LIN {X 0,Y 191.566,Z 1156.427,A -85,B 0,C 180,E1 26720.925,E2 26720.925} C_VEL
LIN {X 0,Y 192.843,Z 1154.444,A -85,B 0,C 180,E1 26730.002,E2 26730.002} C_VEL
LIN {X 0,Y 196.879,Z 1149.231,A -85,B 0,C 180,E1 26741.065,E2 26741.065} C_VEL
LIN {X 0,Y 207.234,Z 1138.669,A -85,B 0,C 180,E1 26753.646,E2 26753.646} C_VEL
LIN {X 0,Y 224.893,Z 1123.007,A -85,B 0,C 180,E1 26764.832,E2 26764.832} C_VEL
LIN {X 0,Y 251.173,Z 1099.179,A -85,B 0,C 180,E1 26774.987,E2 26774.987} C_VEL
LIN {X 0,Y 277.841,Z 1072.352,A -85,B 0,C 180,E1 26782.06,E2 26782.06} C_VEL
LIN {X 0,Y 304.908,Z 1041.471,A -85,B 0,C 180,E1 26787.41,E2 26787.41} C_VEL
LIN {X 0,Y 331.682,Z 1005.034,A -85,B 0,C 180,E1 26791.629,E2 26791.629} C_VEL
LIN {X 0,Y 342.464,Z 988.031,A -85,B 0,C 180,E1 26793.214,E2 26793.214} C_VEL
LIN {X 0,Y 343.901,Z 974.485,A -85,B 0,C 180,E1 26798.43,E2 26798.43} C_VEL
LIN {X 0,Y 344.575,Z 965.223,A -85,B 0,C 180,E1 26803.46,E2 26803.46} C_VEL
LIN {X 0,Y 345.07,Z 960.519,A -85,B 0,C 180,E1 26807.345,E2 26807.345} C_VEL
LIN {X 0,Y 345.918,Z 957.861,A -85,B 0,C 180,E1 26812.462,E2 26812.462} C_VEL
LIN {X 0,Y 347.076,Z 958.983,A -85,B 0,C 180,E1 26817.498,E2 26817.498} C_VEL
LIN {X 0,Y 347.693,Z 967.716,A -85,B 0,C 180,E1 26823.731,E2 26823.731} C_VEL
LIN {X 0,Y 348.349,Z 980.913,A -85,B 0,C 180,E1 26829.355,E2 26829.355} C_VEL
LIN {X 0,Y 347.764,Z 992.361,A -85,B 0,C 180,E1 26832.89,E2 26832.89} C_VEL
LIN {X 0,Y 323.579,Z 1030.844,A -85,B 0,C 180,E1 26836.052,E2 26836.052} C_VEL
LIN {X 0,Y 294.069,Z 1070.126,A -85,B 0,C 180,E1 26840.887,E2 26840.887} C_VEL
LIN {X 0,Y 267.286,Z 1101.116,A -85,B 0,C 180,E1 26846.664,E2 26846.664} C_VEL
LIN {X 0,Y 239.619,Z 1130.083,A -85,B 0,C 180,E1 26854.929,E2 26854.929} C_VEL
LIN {X 0,Y 217.272,Z 1152.485,A -85,B 0,C 180,E1 26865.053,E2 26865.053} C_VEL
LIN {X 0,Y 200.773,Z 1170.696,A -85,B 0,C 180,E1 26878.204,E2 26878.204} C_VEL
LIN {X 0,Y 194.125,Z 1180.088,A -85,B 0,C 180,E1 26889.055,E2 26889.055} C_VEL
LIN {X 0,Y 191.649,Z 1186.194,A -85,B 0,C 180,E1 26900.924,E2 26900.924} C_VEL
LIN {X 0,Y 192.034,Z 1188.018,A -85,B 0,C 180,E1 26909.998,E2 26909.998} C_VEL
LIN {X 0,Y 191.495,Z 1187.446,A -85,B 0,C 180,E1 26919.078,E2 26919.078} C_VEL
LIN {X 0,Y 194.837,Z 1182.07,A -85,B 0,C 180,E1 26932.815,E2 26932.815} C_VEL
LIN {X 0,Y 206.4,Z 1170.637,A -85,B 0,C 180,E1 26947.155,E2 26947.155} C_VEL
